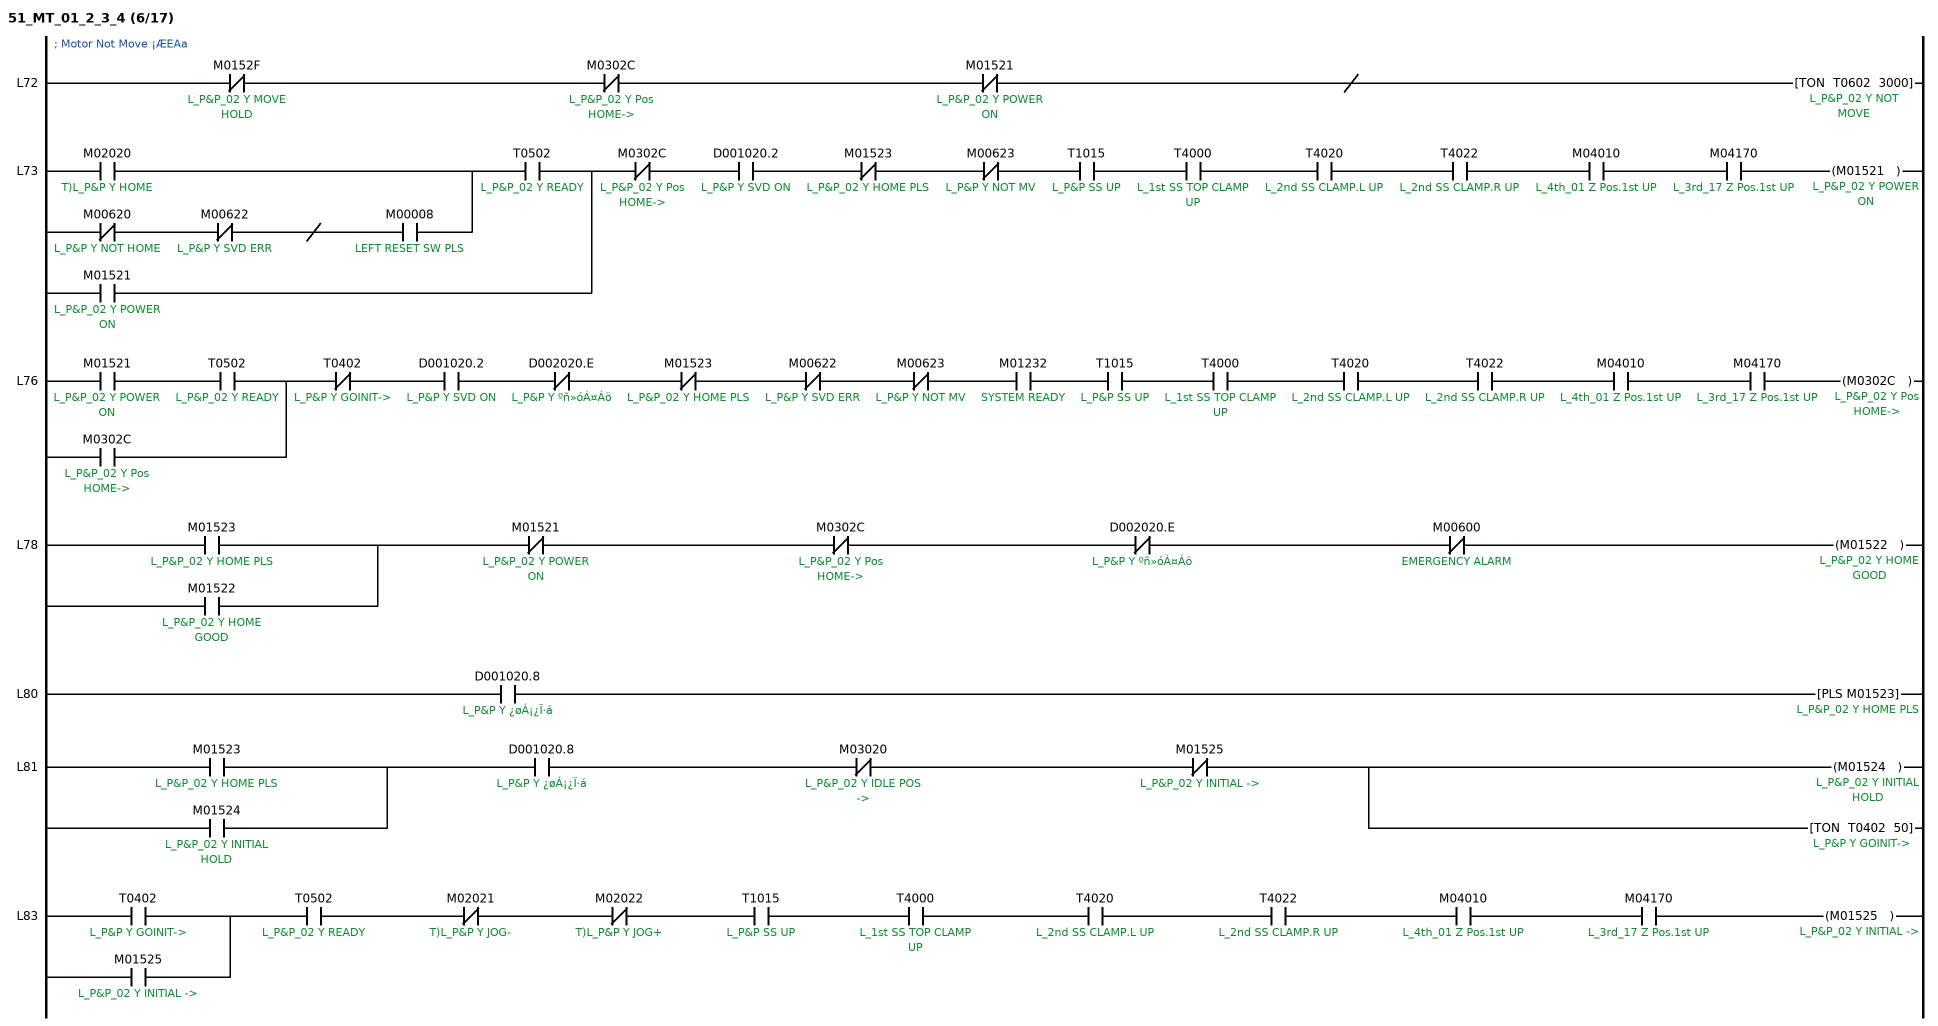
[picture p264: 51_MT_01_2_3_4 rungs L72-L83]
; L72
LOAD NOT  M0152F	// L_P&P_02 Y MOVE HOLD
AND NOT   M0302C	// L_P&P_02 Y Pos HOME->
AND NOT   M01521	// L_P&P_02 Y POWER ON
NOT
TON       T0602 3000	// L_P&P_02 Y NOT MOVE
// output comment: Motor Not Move ¡ÆEAa
; L73
LOAD      M02020	// T)L_P&P Y HOME
LOAD NOT  M00620	// L_P&P Y NOT HOME
AND NOT   M00622	// L_P&P Y SVD ERR
NOT
AND       M00008	// LEFT RESET SW PLS
OR LOAD
AND       T0502	// L_P&P_02 Y READY
OR        M01521	// L_P&P_02 Y POWER ON
AND NOT   M0302C	// L_P&P_02 Y Pos HOME->
AND       D001020.2	// L_P&P Y SVD ON
AND NOT   M01523	// L_P&P_02 Y HOME PLS
AND NOT   M00623	// L_P&P Y NOT MV
AND       T1015	// L_P&P SS UP
AND       T4000	// L_1st SS TOP CLAMP    UP
AND       T4020	// L_2nd SS CLAMP.L UP
AND       T4022	// L_2nd SS CLAMP.R UP
AND       M04010	// L_4th_01 Z Pos.1st UP
AND       M04170	// L_3rd_17 Z Pos.1st UP
OUT       M01521	// L_P&P_02 Y POWER ON
; L76
LOAD      M01521	// L_P&P_02 Y POWER ON
AND       T0502	// L_P&P_02 Y READY
OR        M0302C	// L_P&P_02 Y Pos HOME->
AND NOT   T0402	// L_P&P Y GOINIT->
AND       D001020.2	// L_P&P Y SVD ON
AND NOT   D002020.E	// L_P&P Y ºñ»óÁ¤Áö
AND NOT   M01523	// L_P&P_02 Y HOME PLS
AND NOT   M00622	// L_P&P Y SVD ERR
AND NOT   M00623	// L_P&P Y NOT MV
AND       M01232	// SYSTEM READY
AND       T1015	// L_P&P SS UP
AND       T4000	// L_1st SS TOP CLAMP    UP
AND       T4020	// L_2nd SS CLAMP.L UP
AND       T4022	// L_2nd SS CLAMP.R UP
AND       M04010	// L_4th_01 Z Pos.1st UP
AND       M04170	// L_3rd_17 Z Pos.1st UP
OUT       M0302C	// L_P&P_02 Y Pos HOME->
; L78
LOAD      M01523	// L_P&P_02 Y HOME PLS
OR        M01522	// L_P&P_02 Y HOME GOOD
AND NOT   M01521	// L_P&P_02 Y POWER ON
AND NOT   M0302C	// L_P&P_02 Y Pos HOME->
AND NOT   D002020.E	// L_P&P Y ºñ»óÁ¤Áö
AND NOT   M00600	// EMERGENCY ALARM
OUT       M01522	// L_P&P_02 Y HOME GOOD
; L80
LOAD      D001020.8	// L_P&P Y ¿øÁ¡¿Ï·á
OUTP      M01523	// L_P&P_02 Y HOME PLS
; L81
LOAD      M01523	// L_P&P_02 Y HOME PLS
OR        M01524	// L_P&P_02 Y INITIAL HOLD
AND       D001020.8	// L_P&P Y ¿øÁ¡¿Ï·á
AND NOT   M03020	// L_P&P_02 Y IDLE POS ->
AND NOT   M01525	// L_P&P_02 Y INITIAL ->
OUT       M01524	// L_P&P_02 Y INITIAL HOLD
TON       T0402 50	// L_P&P Y GOINIT->
; L83
LOAD      T0402	// L_P&P Y GOINIT->
OR        M01525	// L_P&P_02 Y INITIAL ->
AND       T0502	// L_P&P_02 Y READY
AND NOT   M02021	// T)L_P&P Y JOG-
AND NOT   M02022	// T)L_P&P Y JOG+
AND       T1015	// L_P&P SS UP
AND       T4000	// L_1st SS TOP CLAMP    UP
AND       T4020	// L_2nd SS CLAMP.L UP
AND       T4022	// L_2nd SS CLAMP.R UP
AND       M04010	// L_4th_01 Z Pos.1st UP
AND       M04170	// L_3rd_17 Z Pos.1st UP
OUT       M01525	// L_P&P_02 Y INITIAL ->

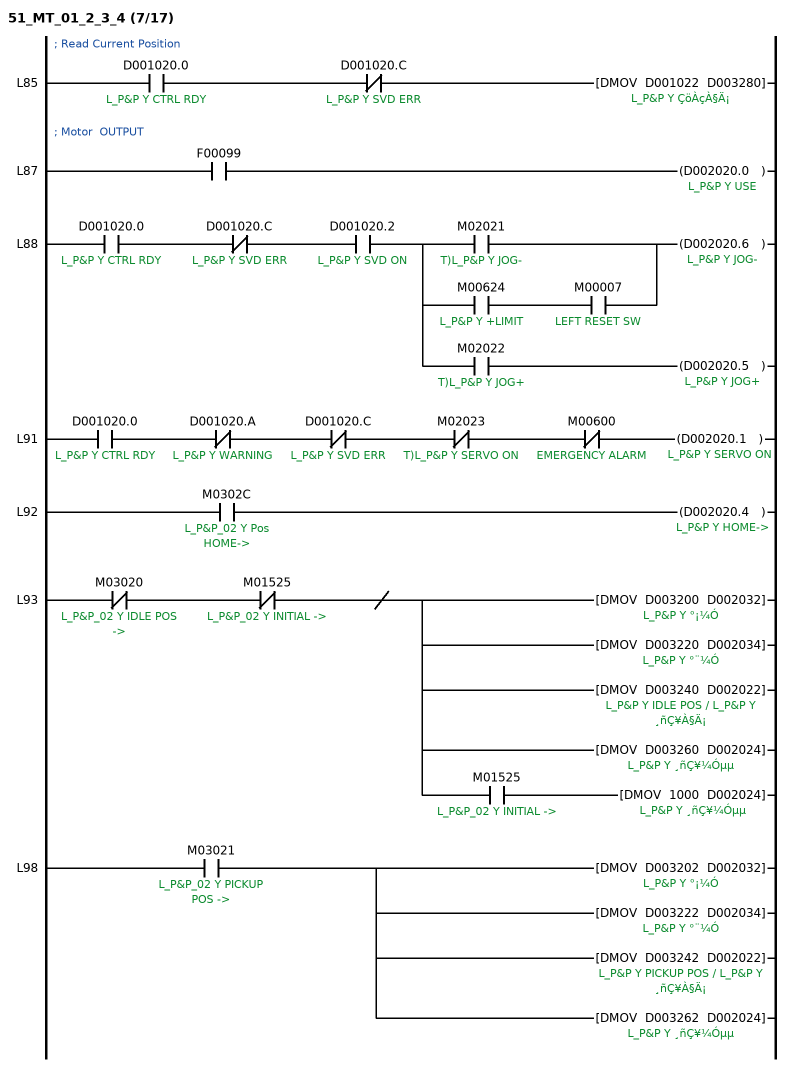
; L85
LOAD      D001020.0	// L_P&P Y CTRL RDY
AND NOT   D001020.C	// L_P&P Y SVD ERR
DMOV      D001022 D003280	// L_P&P Y ÇöÀçÀ§Ä¡
// output comment: Read Current Position
//  Motor  OUTPUT
; L87
LOAD      F00099
OUT       D002020.0	// L_P&P Y USE
; L88
LOAD      D001020.0	// L_P&P Y CTRL RDY
AND NOT   D001020.C	// L_P&P Y SVD ERR
AND       D001020.2	// L_P&P Y SVD ON
MPUSH
LOAD      M02021	// T)L_P&P Y JOG-
LOAD      M00624	// L_P&P Y +LIMIT
AND       M00007	// LEFT RESET SW
OR LOAD
AND LOAD
OUT       D002020.6	// L_P&P Y JOG-
MPOP
AND       M02022	// T)L_P&P Y JOG+
OUT       D002020.5	// L_P&P Y JOG+
; L91
LOAD      D001020.0	// L_P&P Y CTRL RDY
AND NOT   D001020.A	// L_P&P Y WARNING
AND NOT   D001020.C	// L_P&P Y SVD ERR
AND NOT   M02023	// T)L_P&P Y SERVO ON
AND NOT   M00600	// EMERGENCY ALARM
OUT       D002020.1	// L_P&P Y SERVO ON
; L92
LOAD      M0302C	// L_P&P_02 Y Pos HOME->
OUT       D002020.4	// L_P&P Y HOME->
; L93
LOAD NOT  M03020	// L_P&P_02 Y IDLE POS ->
AND NOT   M01525	// L_P&P_02 Y INITIAL ->
NOT
DMOV      D003200 D002032	// L_P&P Y °¡¼Ó
DMOV      D003220 D002034	// L_P&P Y °¨¼Ó
DMOV      D003240 D002022	// L_P&P Y IDLE POS / L_P&P Y ¸ñÇ¥À§Ä¡
DMOV      D003260 D002024	// L_P&P Y ¸ñÇ¥¼Óµµ
AND       M01525	// L_P&P_02 Y INITIAL ->
DMOV      1000 D002024	// L_P&P Y ¸ñÇ¥¼Óµµ
; L98
LOAD      M03021	// L_P&P_02 Y PICKUP POS ->
DMOV      D003202 D002032	// L_P&P Y °¡¼Ó
DMOV      D003222 D002034	// L_P&P Y °¨¼Ó
DMOV      D003242 D002022	// L_P&P Y PICKUP POS / L_P&P Y ¸ñÇ¥À§Ä¡
DMOV      D003262 D002024	// L_P&P Y ¸ñÇ¥¼Óµµ

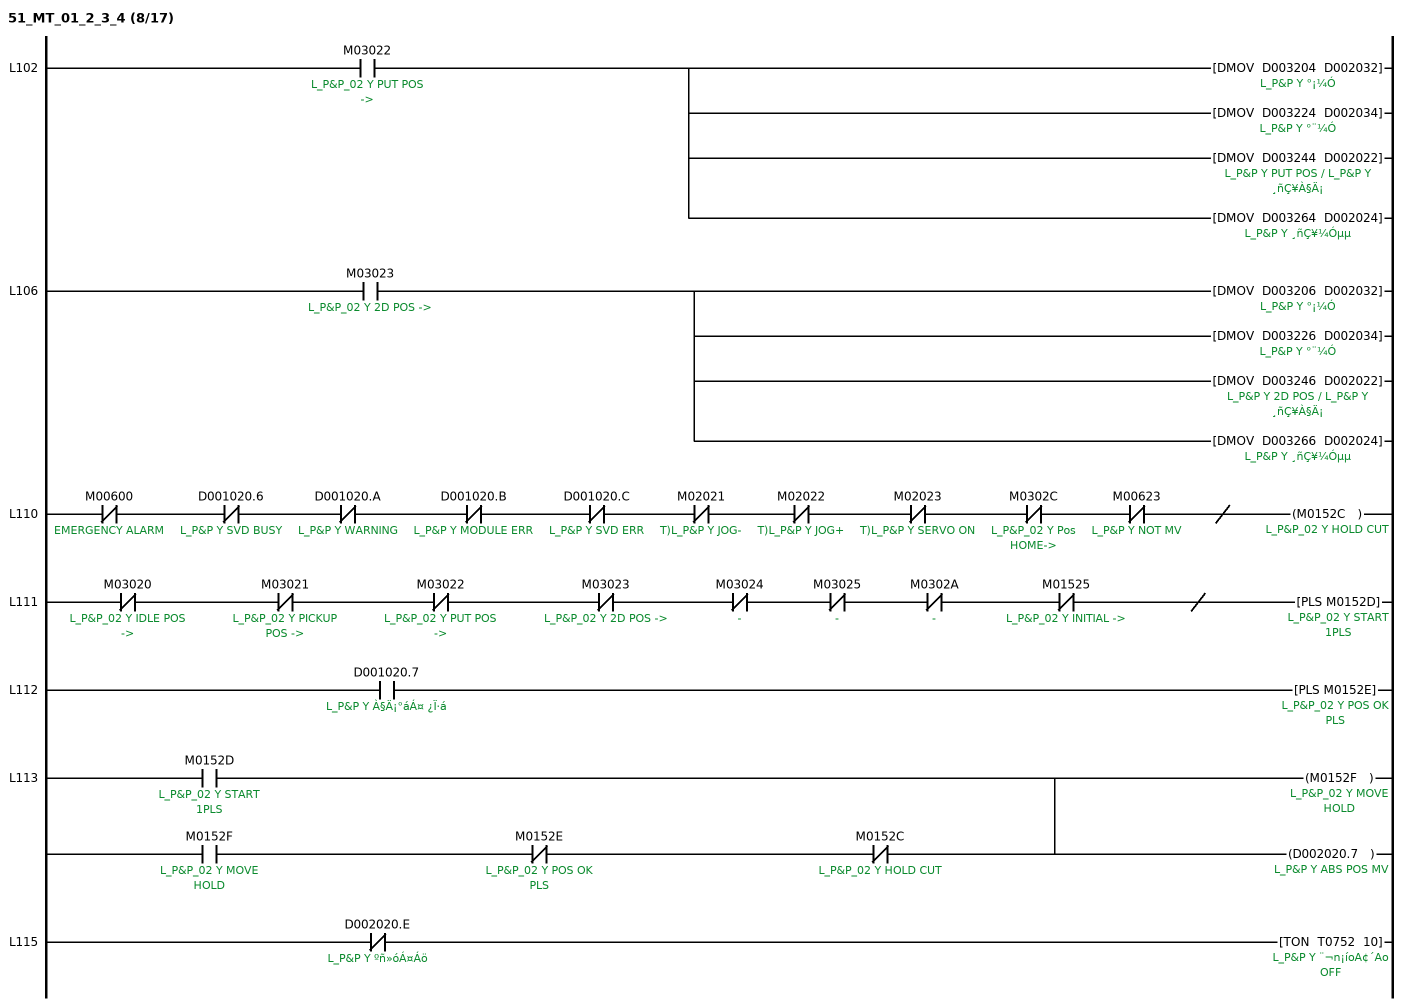
; L102
LOAD      M03022	// L_P&P_02 Y PUT POS ->
DMOV      D003204 D002032	// L_P&P Y °¡¼Ó
DMOV      D003224 D002034	// L_P&P Y °¨¼Ó
DMOV      D003244 D002022	// L_P&P Y PUT POS / L_P&P Y ¸ñÇ¥À§Ä¡
DMOV      D003264 D002024	// L_P&P Y ¸ñÇ¥¼Óµµ
; L106
LOAD      M03023	// L_P&P_02 Y 2D POS ->
DMOV      D003206 D002032	// L_P&P Y °¡¼Ó
DMOV      D003226 D002034	// L_P&P Y °¨¼Ó
DMOV      D003246 D002022	// L_P&P Y 2D POS / L_P&P Y ¸ñÇ¥À§Ä¡
DMOV      D003266 D002024	// L_P&P Y ¸ñÇ¥¼Óµµ
; L110
LOAD NOT  M00600	// EMERGENCY ALARM
AND NOT   D001020.6	// L_P&P Y SVD BUSY
AND NOT   D001020.A	// L_P&P Y WARNING
AND NOT   D001020.B	// L_P&P Y MODULE ERR
AND NOT   D001020.C	// L_P&P Y SVD ERR
AND NOT   M02021	// T)L_P&P Y JOG-
AND NOT   M02022	// T)L_P&P Y JOG+
AND NOT   M02023	// T)L_P&P Y SERVO ON
AND NOT   M0302C	// L_P&P_02 Y Pos HOME->
AND NOT   M00623	// L_P&P Y NOT MV
NOT
OUT       M0152C	// L_P&P_02 Y HOLD CUT
; L111
LOAD NOT  M03020	// L_P&P_02 Y IDLE POS ->
AND NOT   M03021	// L_P&P_02 Y PICKUP POS ->
AND NOT   M03022	// L_P&P_02 Y PUT POS ->
AND NOT   M03023	// L_P&P_02 Y 2D POS ->
AND NOT   M03024	// -
AND NOT   M03025	// -
AND NOT   M0302A	// -
AND NOT   M01525	// L_P&P_02 Y INITIAL ->
NOT
OUTP      M0152D	// L_P&P_02 Y START 1PLS
; L112
LOAD      D001020.7	// L_P&P Y À§Ä¡°áÁ¤ ¿Ï·á
OUTP      M0152E	// L_P&P_02 Y POS OK PLS
; L113
LOAD      M0152D	// L_P&P_02 Y START 1PLS
LOAD      M0152F	// L_P&P_02 Y MOVE HOLD
AND NOT   M0152E	// L_P&P_02 Y POS OK PLS
AND NOT   M0152C	// L_P&P_02 Y HOLD CUT
OR LOAD
OUT       M0152F	// L_P&P_02 Y MOVE HOLD
OUT       D002020.7	// L_P&P Y ABS POS MV
; L115
LOAD NOT  D002020.E	// L_P&P Y ºñ»óÁ¤Áö
TON       T0752 10	// L_P&P Y ¨¬n¡íoA¢´AoOFF

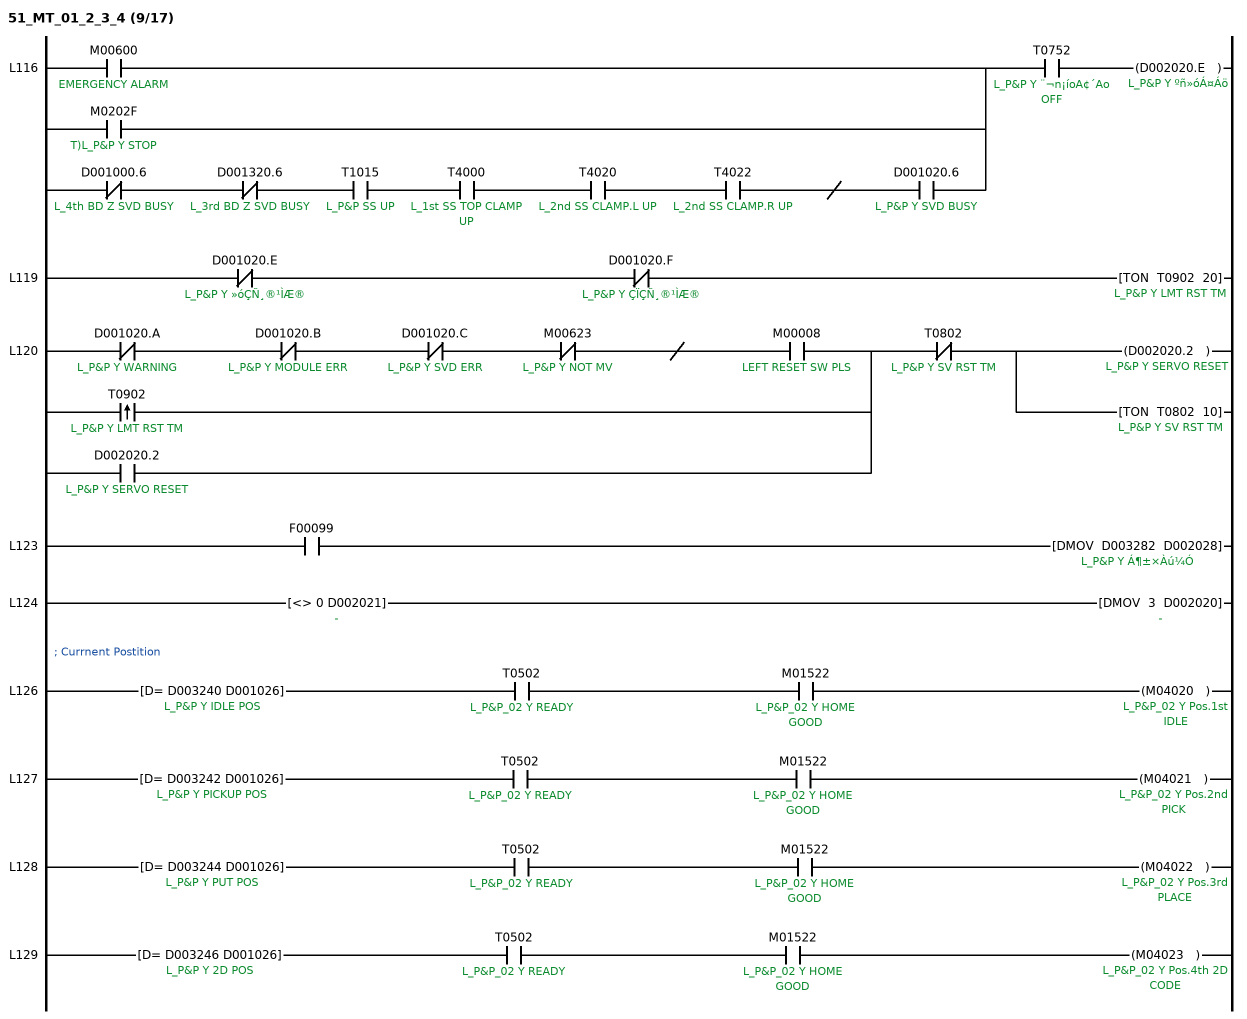
; L116
LOAD      M00600	// EMERGENCY ALARM
OR        M0202F	// T)L_P&P Y STOP
LOAD NOT  D001000.6	// L_4th BD Z SVD BUSY
AND NOT   D001320.6	// L_3rd BD Z SVD BUSY
AND       T1015	// L_P&P SS UP
AND       T4000	// L_1st SS TOP CLAMP    UP
AND       T4020	// L_2nd SS CLAMP.L UP
AND       T4022	// L_2nd SS CLAMP.R UP
NOT
AND       D001020.6	// L_P&P Y SVD BUSY
OR LOAD
AND       T0752	// L_P&P Y ¨¬n¡íoA¢´AoOFF
OUT       D002020.E	// L_P&P Y ºñ»óÁ¤Áö
; L119
LOAD NOT  D001020.E	// L_P&P Y »óÇÑ¸®¹ÌÆ®
AND NOT   D001020.F	// L_P&P Y ÇÏÇÑ¸®¹ÌÆ®
TON       T0902 20	// L_P&P Y LMT RST TM
; L120
LOAD NOT  D001020.A	// L_P&P Y WARNING
AND NOT   D001020.B	// L_P&P Y MODULE ERR
AND NOT   D001020.C	// L_P&P Y SVD ERR
AND NOT   M00623	// L_P&P Y NOT MV
NOT
AND       M00008	// LEFT RESET SW PLS
ORP       T0902	// L_P&P Y LMT RST TM
OR        D002020.2	// L_P&P Y SERVO RESET
AND NOT   T0802	// L_P&P Y SV RST TM
OUT       D002020.2	// L_P&P Y SERVO RESET
TON       T0802 10	// L_P&P Y SV RST TM
; L123
LOAD      F00099
DMOV      D003282 D002028	// L_P&P Y Á¶±×Àú¼Ó
; L124
LOAD<>    0 D002021	// -
DMOV      3 D002020	// -
// Currnent Postition
; L126
LOADD=    D003240 D001026	// L_P&P Y IDLE POS
AND       T0502	// L_P&P_02 Y READY
AND       M01522	// L_P&P_02 Y HOME GOOD
OUT       M04020	// L_P&P_02 Y Pos.1st IDLE
; L127
LOADD=    D003242 D001026	// L_P&P Y PICKUP POS
AND       T0502	// L_P&P_02 Y READY
AND       M01522	// L_P&P_02 Y HOME GOOD
OUT       M04021	// L_P&P_02 Y Pos.2nd PICK
; L128
LOADD=    D003244 D001026	// L_P&P Y PUT POS
AND       T0502	// L_P&P_02 Y READY
AND       M01522	// L_P&P_02 Y HOME GOOD
OUT       M04022	// L_P&P_02 Y Pos.3rd PLACE
; L129
LOADD=    D003246 D001026	// L_P&P Y 2D POS
AND       T0502	// L_P&P_02 Y READY
AND       M01522	// L_P&P_02 Y HOME GOOD
OUT       M04023	// L_P&P_02 Y Pos.4th 2D CODE

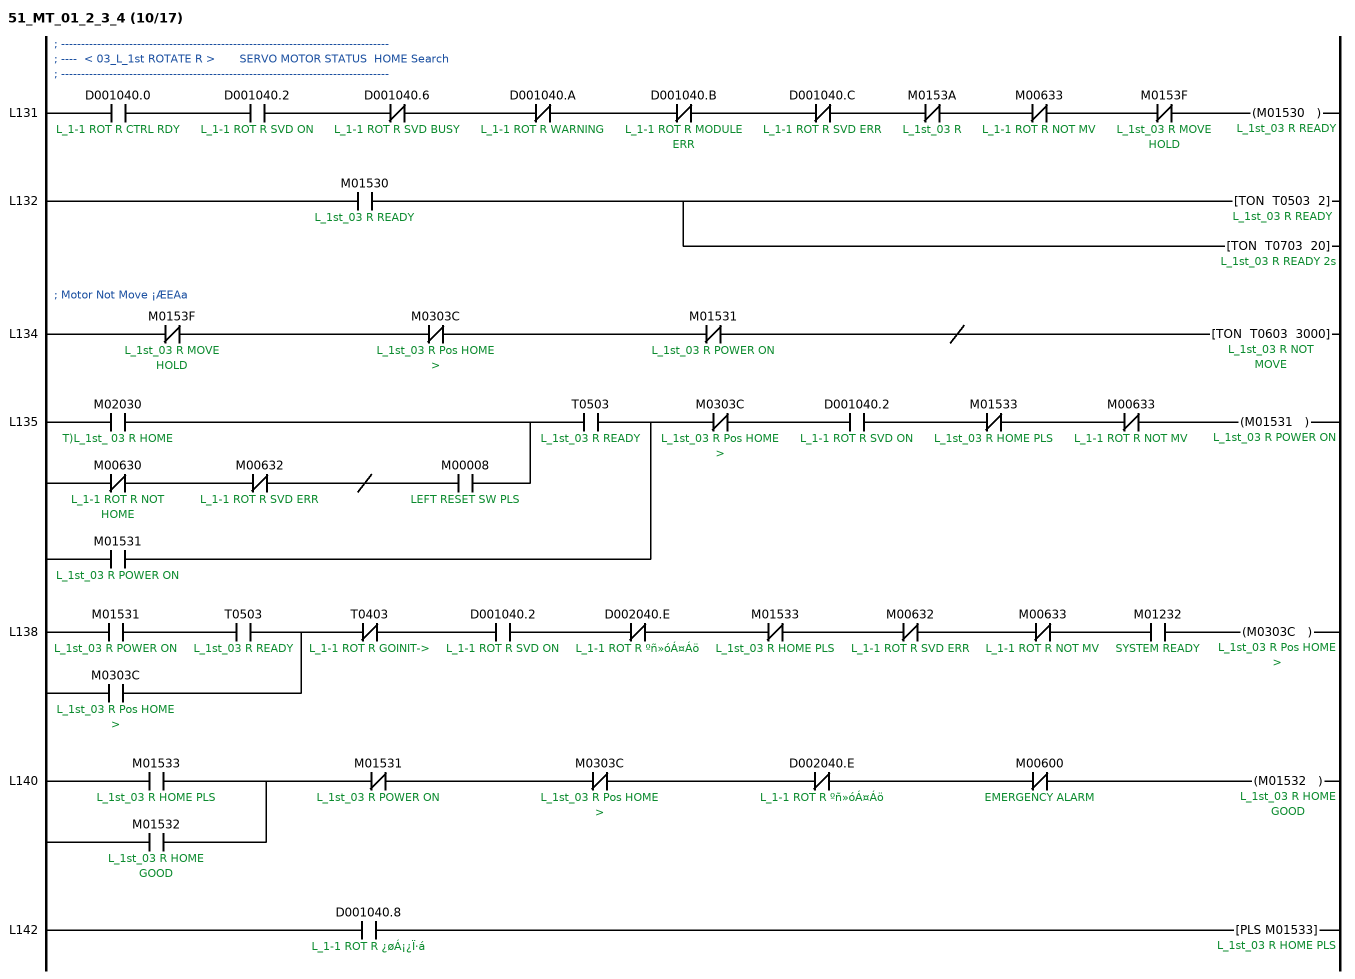
// ----------------------------------------------------------------------------------
// 
// ----  < 03_L_1st ROTATE R >       SERVO MOTOR STATUS  HOME Search
// 
// ----------------------------------------------------------------------------------
; L131
LOAD      D001040.0	// L_1-1 ROT R CTRL RDY
AND       D001040.2	// L_1-1 ROT R SVD ON
AND NOT   D001040.6	// L_1-1 ROT R SVD BUSY
AND NOT   D001040.A	// L_1-1 ROT R WARNING
AND NOT   D001040.B	// L_1-1 ROT R MODULE ERR
AND NOT   D001040.C	// L_1-1 ROT R SVD ERR
AND NOT   M0153A	// L_1st_03 R
AND NOT   M00633	// L_1-1 ROT R NOT MV
AND NOT   M0153F	// L_1st_03 R MOVE HOLD
OUT       M01530	// L_1st_03 R READY
; L132
LOAD      M01530	// L_1st_03 R READY
TON       T0503 2	// L_1st_03 R READY
TON       T0703 20	// L_1st_03 R READY 2s
; L134
LOAD NOT  M0153F	// L_1st_03 R MOVE HOLD
AND NOT   M0303C	// L_1st_03 R Pos HOME >
AND NOT   M01531	// L_1st_03 R POWER ON
NOT
TON       T0603 3000	// L_1st_03 R NOT MOVE
// output comment: Motor Not Move ¡ÆEAa
; L135
LOAD      M02030	// T)L_1st_ 03 R HOME
LOAD NOT  M00630	// L_1-1 ROT R NOT HOME
AND NOT   M00632	// L_1-1 ROT R SVD ERR
NOT
AND       M00008	// LEFT RESET SW PLS
OR LOAD
AND       T0503	// L_1st_03 R READY
OR        M01531	// L_1st_03 R POWER ON
AND NOT   M0303C	// L_1st_03 R Pos HOME >
AND       D001040.2	// L_1-1 ROT R SVD ON
AND NOT   M01533	// L_1st_03 R HOME PLS
AND NOT   M00633	// L_1-1 ROT R NOT MV
OUT       M01531	// L_1st_03 R POWER ON
; L138
LOAD      M01531	// L_1st_03 R POWER ON
AND       T0503	// L_1st_03 R READY
OR        M0303C	// L_1st_03 R Pos HOME >
AND NOT   T0403	// L_1-1 ROT R GOINIT->
AND       D001040.2	// L_1-1 ROT R SVD ON
AND NOT   D002040.E	// L_1-1 ROT R ºñ»óÁ¤Áö
AND NOT   M01533	// L_1st_03 R HOME PLS
AND NOT   M00632	// L_1-1 ROT R SVD ERR
AND NOT   M00633	// L_1-1 ROT R NOT MV
AND       M01232	// SYSTEM READY
OUT       M0303C	// L_1st_03 R Pos HOME >
; L140
LOAD      M01533	// L_1st_03 R HOME PLS
OR        M01532	// L_1st_03 R HOME GOOD
AND NOT   M01531	// L_1st_03 R POWER ON
AND NOT   M0303C	// L_1st_03 R Pos HOME >
AND NOT   D002040.E	// L_1-1 ROT R ºñ»óÁ¤Áö
AND NOT   M00600	// EMERGENCY ALARM
OUT       M01532	// L_1st_03 R HOME GOOD
; L142
LOAD      D001040.8	// L_1-1 ROT R ¿øÁ¡¿Ï·á
OUTP      M01533	// L_1st_03 R HOME PLS

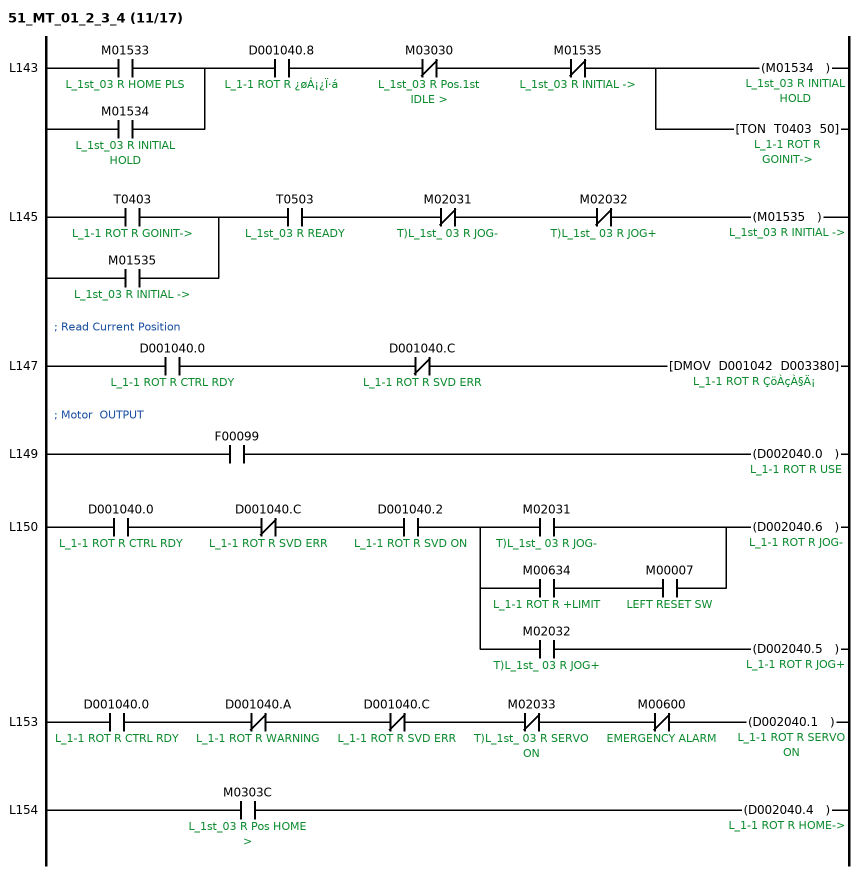
; L143
LOAD      M01533	// L_1st_03 R HOME PLS
OR        M01534	// L_1st_03 R INITIAL HOLD
AND       D001040.8	// L_1-1 ROT R ¿øÁ¡¿Ï·á
AND NOT   M03030	// L_1st_03 R Pos.1st IDLE >
AND NOT   M01535	// L_1st_03 R INITIAL ->
OUT       M01534	// L_1st_03 R INITIAL HOLD
TON       T0403 50	// L_1-1 ROT R GOINIT->
; L145
LOAD      T0403	// L_1-1 ROT R GOINIT->
OR        M01535	// L_1st_03 R INITIAL ->
AND       T0503	// L_1st_03 R READY
AND NOT   M02031	// T)L_1st_ 03 R JOG-
AND NOT   M02032	// T)L_1st_ 03 R JOG+
OUT       M01535	// L_1st_03 R INITIAL ->
; L147
LOAD      D001040.0	// L_1-1 ROT R CTRL RDY
AND NOT   D001040.C	// L_1-1 ROT R SVD ERR
DMOV      D001042 D003380	// L_1-1 ROT R ÇöÀçÀ§Ä¡
// output comment: Read Current Position
//  Motor  OUTPUT
; L149
LOAD      F00099
OUT       D002040.0	// L_1-1 ROT R USE
; L150
LOAD      D001040.0	// L_1-1 ROT R CTRL RDY
AND NOT   D001040.C	// L_1-1 ROT R SVD ERR
AND       D001040.2	// L_1-1 ROT R SVD ON
MPUSH
LOAD      M02031	// T)L_1st_ 03 R JOG-
LOAD      M00634	// L_1-1 ROT R +LIMIT
AND       M00007	// LEFT RESET SW
OR LOAD
AND LOAD
OUT       D002040.6	// L_1-1 ROT R JOG-
MPOP
AND       M02032	// T)L_1st_ 03 R JOG+
OUT       D002040.5	// L_1-1 ROT R JOG+
; L153
LOAD      D001040.0	// L_1-1 ROT R CTRL RDY
AND NOT   D001040.A	// L_1-1 ROT R WARNING
AND NOT   D001040.C	// L_1-1 ROT R SVD ERR
AND NOT   M02033	// T)L_1st_ 03 R SERVO ON
AND NOT   M00600	// EMERGENCY ALARM
OUT       D002040.1	// L_1-1 ROT R SERVO ON
; L154
LOAD      M0303C	// L_1st_03 R Pos HOME >
OUT       D002040.4	// L_1-1 ROT R HOME->

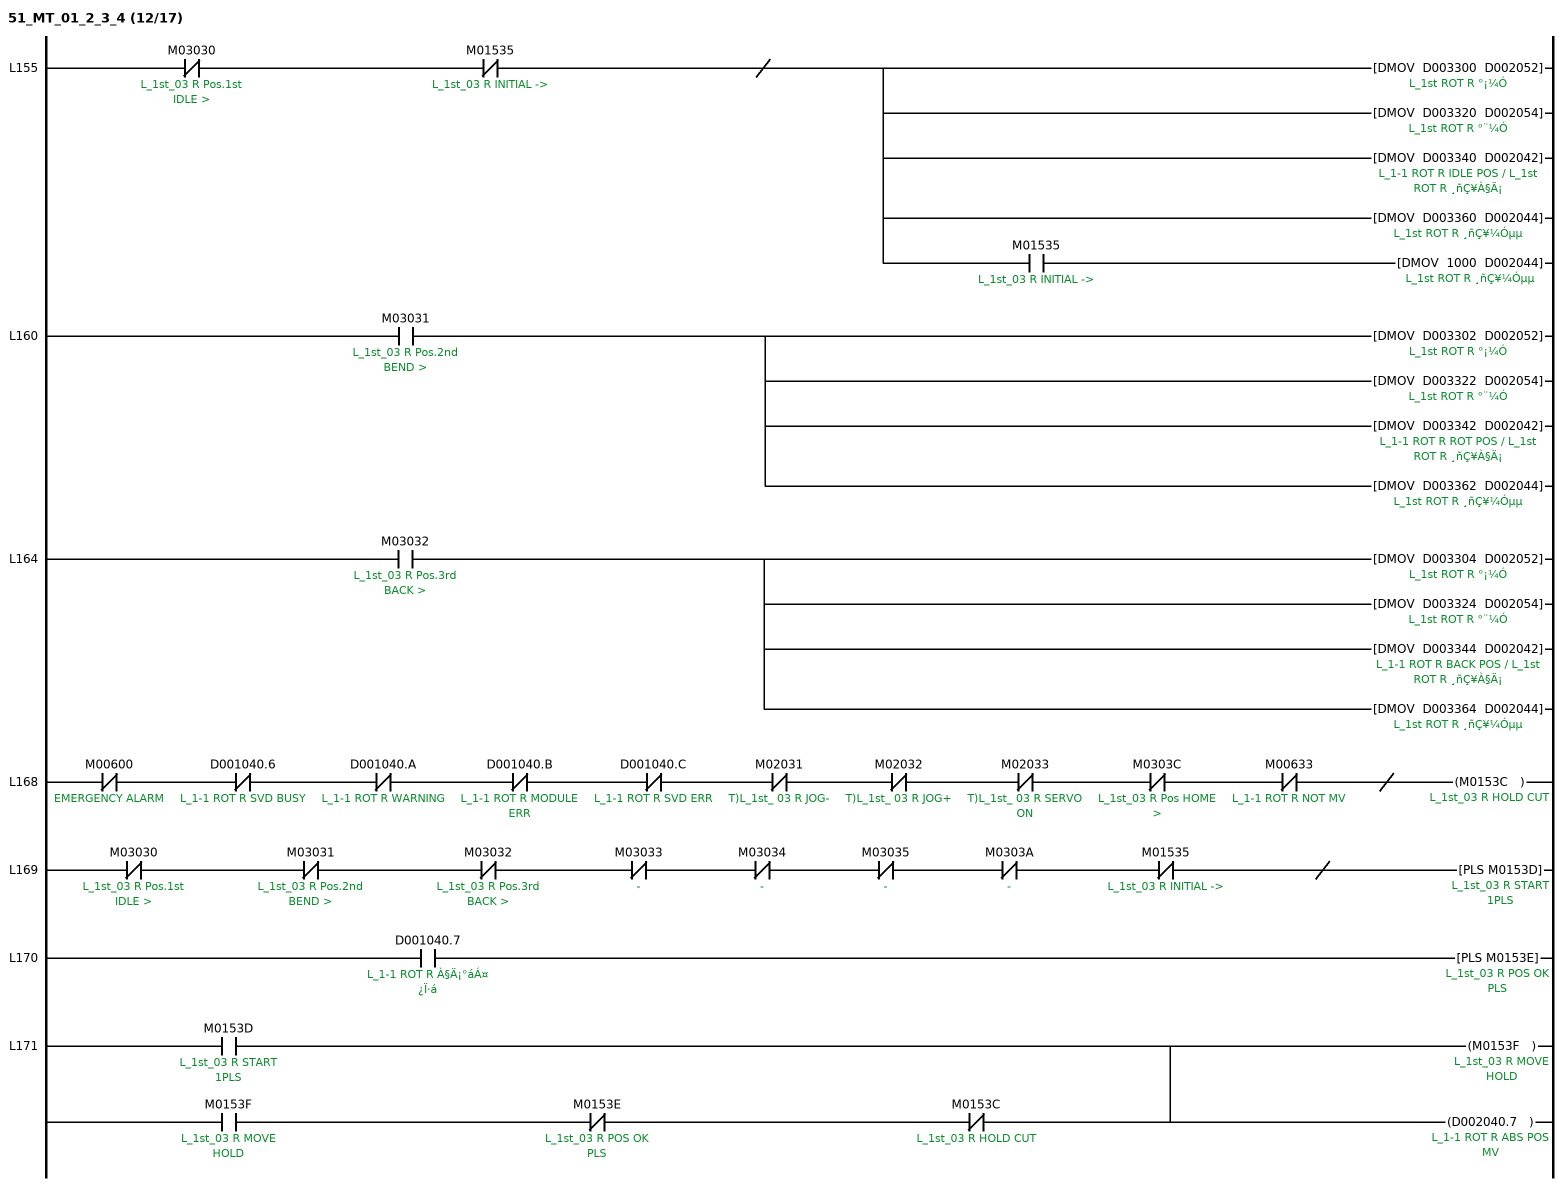
; L155
LOAD NOT  M03030	// L_1st_03 R Pos.1st IDLE >
AND NOT   M01535	// L_1st_03 R INITIAL ->
NOT
DMOV      D003300 D002052	// L_1st ROT R °¡¼Ó
DMOV      D003320 D002054	// L_1st ROT R °¨¼Ó
DMOV      D003340 D002042	// L_1-1 ROT R IDLE POS / L_1st ROT R ¸ñÇ¥À§Ä¡
DMOV      D003360 D002044	// L_1st ROT R ¸ñÇ¥¼Óµµ
AND       M01535	// L_1st_03 R INITIAL ->
DMOV      1000 D002044	// L_1st ROT R ¸ñÇ¥¼Óµµ
; L160
LOAD      M03031	// L_1st_03 R Pos.2nd BEND >
DMOV      D003302 D002052	// L_1st ROT R °¡¼Ó
DMOV      D003322 D002054	// L_1st ROT R °¨¼Ó
DMOV      D003342 D002042	// L_1-1 ROT R ROT POS / L_1st ROT R ¸ñÇ¥À§Ä¡
DMOV      D003362 D002044	// L_1st ROT R ¸ñÇ¥¼Óµµ
; L164
LOAD      M03032	// L_1st_03 R Pos.3rd BACK >
DMOV      D003304 D002052	// L_1st ROT R °¡¼Ó
DMOV      D003324 D002054	// L_1st ROT R °¨¼Ó
DMOV      D003344 D002042	// L_1-1 ROT R BACK POS / L_1st ROT R ¸ñÇ¥À§Ä¡
DMOV      D003364 D002044	// L_1st ROT R ¸ñÇ¥¼Óµµ
; L168
LOAD NOT  M00600	// EMERGENCY ALARM
AND NOT   D001040.6	// L_1-1 ROT R SVD BUSY
AND NOT   D001040.A	// L_1-1 ROT R WARNING
AND NOT   D001040.B	// L_1-1 ROT R MODULE ERR
AND NOT   D001040.C	// L_1-1 ROT R SVD ERR
AND NOT   M02031	// T)L_1st_ 03 R JOG-
AND NOT   M02032	// T)L_1st_ 03 R JOG+
AND NOT   M02033	// T)L_1st_ 03 R SERVO ON
AND NOT   M0303C	// L_1st_03 R Pos HOME >
AND NOT   M00633	// L_1-1 ROT R NOT MV
NOT
OUT       M0153C	// L_1st_03 R HOLD CUT
; L169
LOAD NOT  M03030	// L_1st_03 R Pos.1st IDLE >
AND NOT   M03031	// L_1st_03 R Pos.2nd BEND >
AND NOT   M03032	// L_1st_03 R Pos.3rd BACK >
AND NOT   M03033	// -
AND NOT   M03034	// -
AND NOT   M03035	// -
AND NOT   M0303A	// -
AND NOT   M01535	// L_1st_03 R INITIAL ->
NOT
OUTP      M0153D	// L_1st_03 R START 1PLS
; L170
LOAD      D001040.7	// L_1-1 ROT R À§Ä¡°áÁ¤ ¿Ï·á
OUTP      M0153E	// L_1st_03 R POS OK PLS
; L171
LOAD      M0153D	// L_1st_03 R START 1PLS
LOAD      M0153F	// L_1st_03 R MOVE HOLD
AND NOT   M0153E	// L_1st_03 R POS OK PLS
AND NOT   M0153C	// L_1st_03 R HOLD CUT
OR LOAD
OUT       M0153F	// L_1st_03 R MOVE HOLD
OUT       D002040.7	// L_1-1 ROT R ABS POS MV

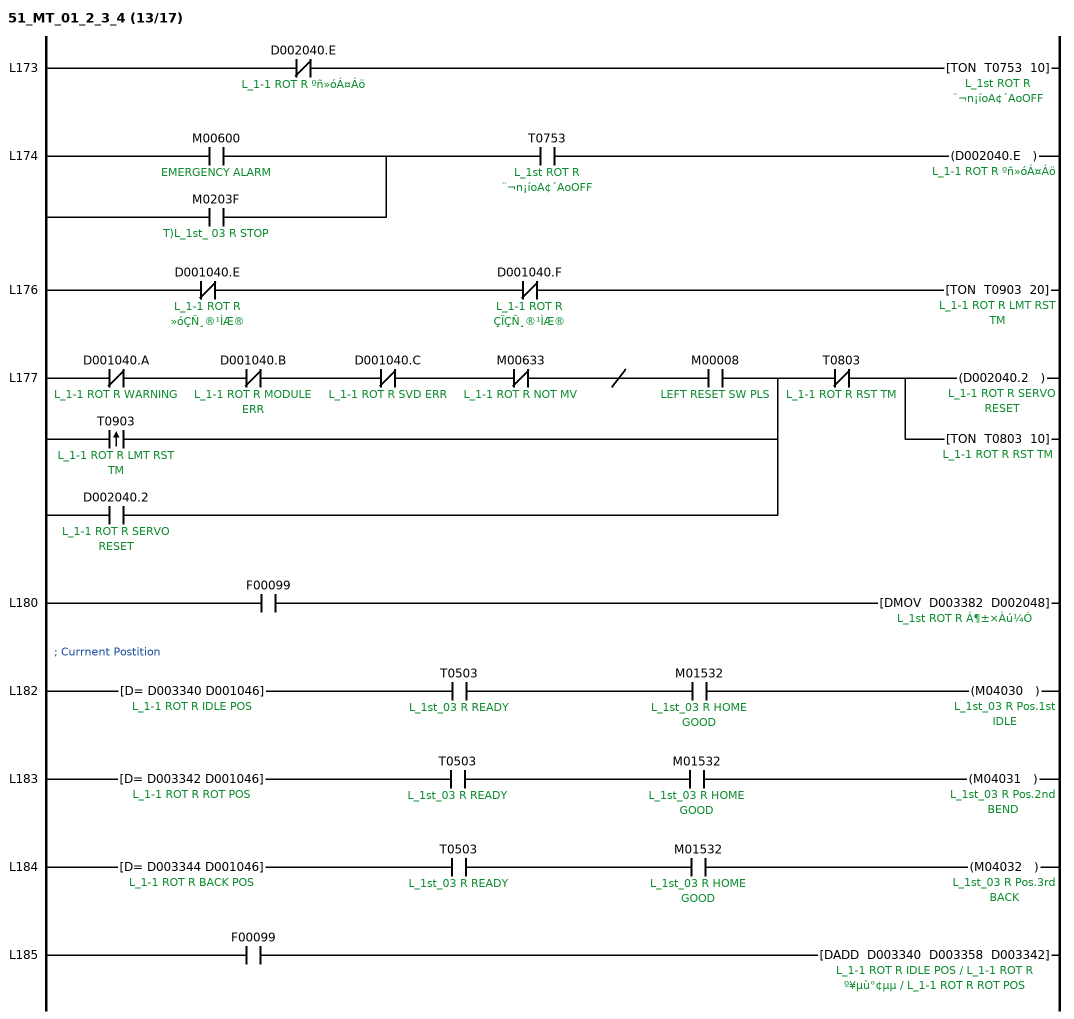
; L173
LOAD NOT  D002040.E	// L_1-1 ROT R ºñ»óÁ¤Áö
TON       T0753 10	// L_1st ROT R ¨¬n¡íoA¢´AoOFF
; L174
LOAD      M00600	// EMERGENCY ALARM
OR        M0203F	// T)L_1st_ 03 R STOP
AND       T0753	// L_1st ROT R ¨¬n¡íoA¢´AoOFF
OUT       D002040.E	// L_1-1 ROT R ºñ»óÁ¤Áö
; L176
LOAD NOT  D001040.E	// L_1-1 ROT R »óÇÑ¸®¹ÌÆ®
AND NOT   D001040.F	// L_1-1 ROT R ÇÏÇÑ¸®¹ÌÆ®
TON       T0903 20	// L_1-1 ROT R LMT RST TM
; L177
LOAD NOT  D001040.A	// L_1-1 ROT R WARNING
AND NOT   D001040.B	// L_1-1 ROT R MODULE ERR
AND NOT   D001040.C	// L_1-1 ROT R SVD ERR
AND NOT   M00633	// L_1-1 ROT R NOT MV
NOT
AND       M00008	// LEFT RESET SW PLS
ORP       T0903	// L_1-1 ROT R LMT RST TM
OR        D002040.2	// L_1-1 ROT R SERVO RESET
AND NOT   T0803	// L_1-1 ROT R RST TM
OUT       D002040.2	// L_1-1 ROT R SERVO RESET
TON       T0803 10	// L_1-1 ROT R RST TM
; L180
LOAD      F00099
DMOV      D003382 D002048	// L_1st ROT R Á¶±×Àú¼Ó
// Currnent Postition
; L182
LOADD=    D003340 D001046	// L_1-1 ROT R IDLE POS
AND       T0503	// L_1st_03 R READY
AND       M01532	// L_1st_03 R HOME GOOD
OUT       M04030	// L_1st_03 R Pos.1st IDLE
; L183
LOADD=    D003342 D001046	// L_1-1 ROT R ROT POS
AND       T0503	// L_1st_03 R READY
AND       M01532	// L_1st_03 R HOME GOOD
OUT       M04031	// L_1st_03 R Pos.2nd BEND
; L184
LOADD=    D003344 D001046	// L_1-1 ROT R BACK POS
AND       T0503	// L_1st_03 R READY
AND       M01532	// L_1st_03 R HOME GOOD
OUT       M04032	// L_1st_03 R Pos.3rd BACK
; L185
LOAD      F00099
DADD      D003340 D003358 D003342	// L_1-1 ROT R IDLE POS / L_1-1 ROT R º¥µù°¢µµ / L_1-1 ROT R ROT POS

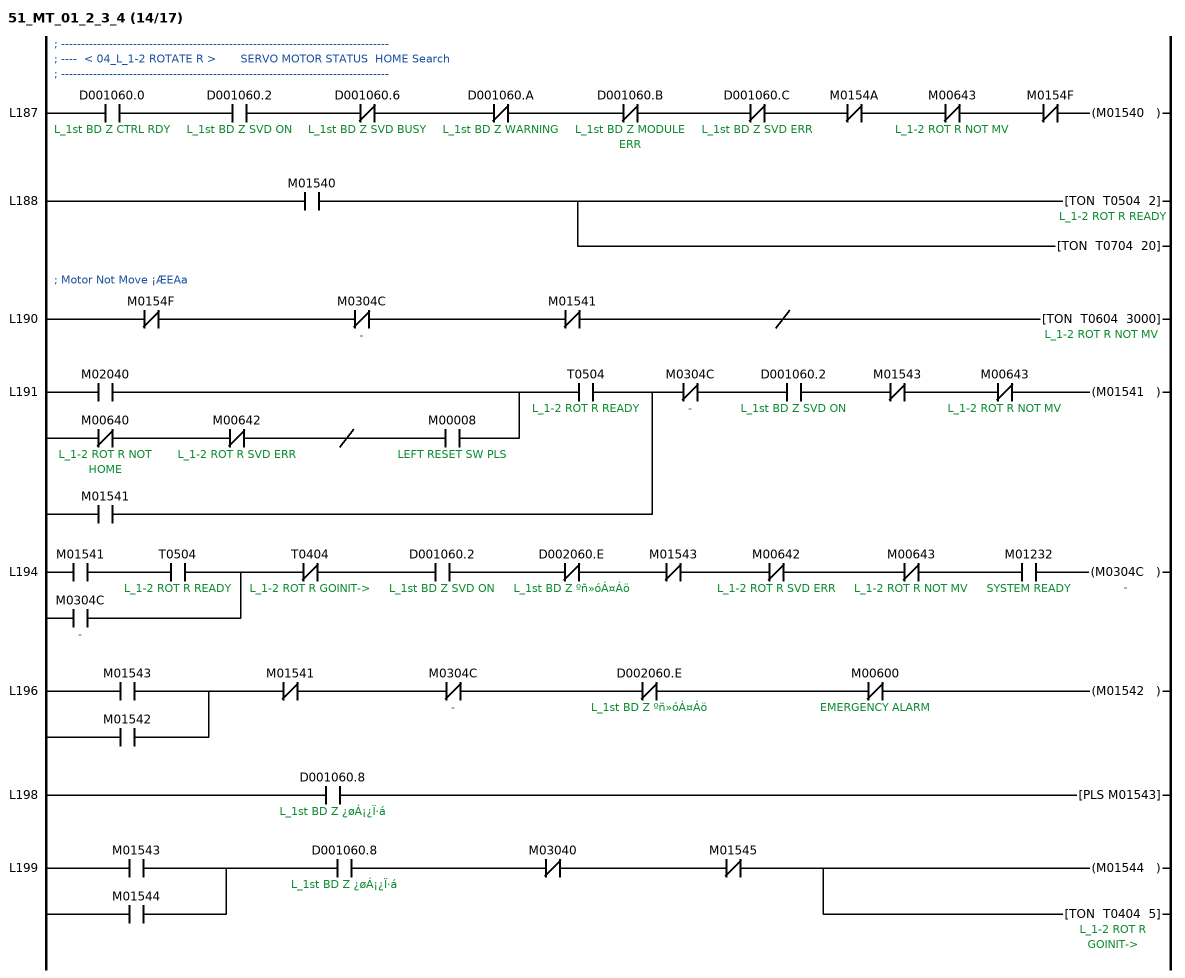
// ----------------------------------------------------------------------------------
// 
// ----  < 04_L_1-2 ROTATE R >       SERVO MOTOR STATUS  HOME Search
// 
// ----------------------------------------------------------------------------------
; L187
LOAD      D001060.0	// L_1st BD Z CTRL RDY
AND       D001060.2	// L_1st BD Z SVD ON
AND NOT   D001060.6	// L_1st BD Z SVD BUSY
AND NOT   D001060.A	// L_1st BD Z WARNING
AND NOT   D001060.B	// L_1st BD Z MODULE ERR
AND NOT   D001060.C	// L_1st BD Z SVD ERR
AND NOT   M0154A
AND NOT   M00643	// L_1-2 ROT R NOT MV
AND NOT   M0154F
OUT       M01540
; L188
LOAD      M01540
TON       T0504 2	// L_1-2 ROT R READY
TON       T0704 20
; L190
LOAD NOT  M0154F
AND NOT   M0304C	// -
AND NOT   M01541
NOT
TON       T0604 3000	// L_1-2 ROT R NOT MV
// output comment: Motor Not Move ¡ÆEAa
; L191
LOAD      M02040
LOAD NOT  M00640	// L_1-2 ROT R NOT HOME
AND NOT   M00642	// L_1-2 ROT R SVD ERR
NOT
AND       M00008	// LEFT RESET SW PLS
OR LOAD
AND       T0504	// L_1-2 ROT R READY
OR        M01541
AND NOT   M0304C	// -
AND       D001060.2	// L_1st BD Z SVD ON
AND NOT   M01543
AND NOT   M00643	// L_1-2 ROT R NOT MV
OUT       M01541
; L194
LOAD      M01541
AND       T0504	// L_1-2 ROT R READY
OR        M0304C	// -
AND NOT   T0404	// L_1-2 ROT R GOINIT->
AND       D001060.2	// L_1st BD Z SVD ON
AND NOT   D002060.E	// L_1st BD Z ºñ»óÁ¤Áö
AND NOT   M01543
AND NOT   M00642	// L_1-2 ROT R SVD ERR
AND NOT   M00643	// L_1-2 ROT R NOT MV
AND       M01232	// SYSTEM READY
OUT       M0304C	// -
; L196
LOAD      M01543
OR        M01542
AND NOT   M01541
AND NOT   M0304C	// -
AND NOT   D002060.E	// L_1st BD Z ºñ»óÁ¤Áö
AND NOT   M00600	// EMERGENCY ALARM
OUT       M01542
; L198
LOAD      D001060.8	// L_1st BD Z ¿øÁ¡¿Ï·á
OUTP      M01543
; L199
LOAD      M01543
OR        M01544
AND       D001060.8	// L_1st BD Z ¿øÁ¡¿Ï·á
AND NOT   M03040
AND NOT   M01545
OUT       M01544
TON       T0404 5	// L_1-2 ROT R GOINIT->

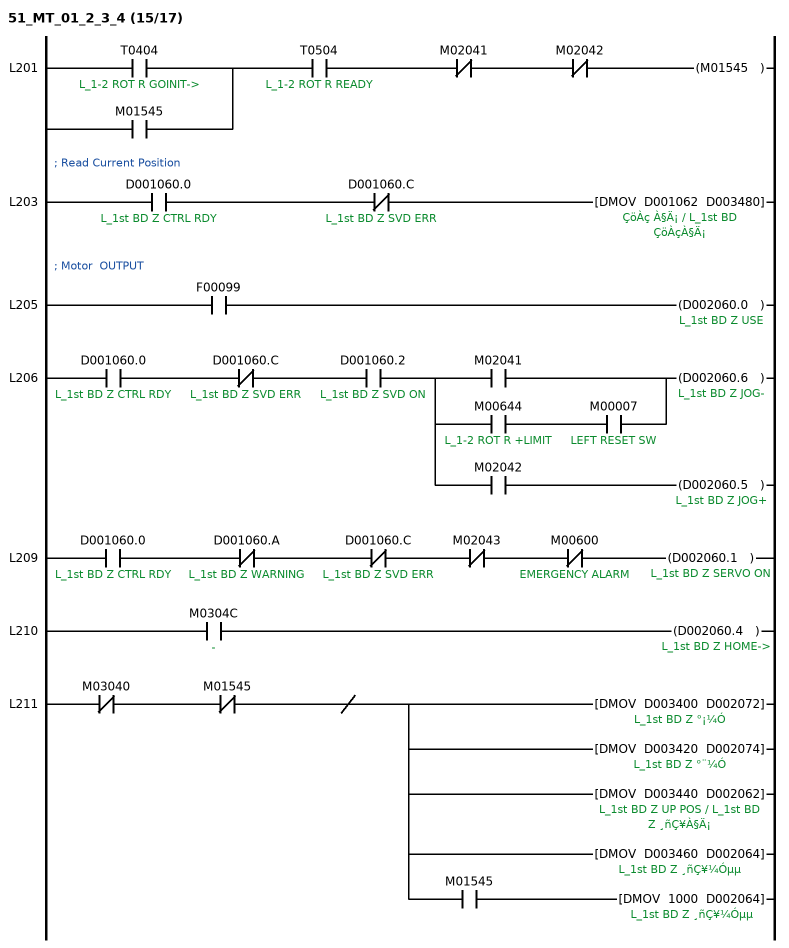
; L201
LOAD      T0404	// L_1-2 ROT R GOINIT->
OR        M01545
AND       T0504	// L_1-2 ROT R READY
AND NOT   M02041
AND NOT   M02042
OUT       M01545
; L203
LOAD      D001060.0	// L_1st BD Z CTRL RDY
AND NOT   D001060.C	// L_1st BD Z SVD ERR
DMOV      D001062 D003480	// ÇöÀç À§Ä¡ / L_1st BD ÇöÀçÀ§Ä¡
// output comment: Read Current Position
//  Motor  OUTPUT
; L205
LOAD      F00099
OUT       D002060.0	// L_1st BD Z USE
; L206
LOAD      D001060.0	// L_1st BD Z CTRL RDY
AND NOT   D001060.C	// L_1st BD Z SVD ERR
AND       D001060.2	// L_1st BD Z SVD ON
MPUSH
LOAD      M02041
LOAD      M00644	// L_1-2 ROT R +LIMIT
AND       M00007	// LEFT RESET SW
OR LOAD
AND LOAD
OUT       D002060.6	// L_1st BD Z JOG-
MPOP
AND       M02042
OUT       D002060.5	// L_1st BD Z JOG+
; L209
LOAD      D001060.0	// L_1st BD Z CTRL RDY
AND NOT   D001060.A	// L_1st BD Z WARNING
AND NOT   D001060.C	// L_1st BD Z SVD ERR
AND NOT   M02043
AND NOT   M00600	// EMERGENCY ALARM
OUT       D002060.1	// L_1st BD Z SERVO ON
; L210
LOAD      M0304C	// -
OUT       D002060.4	// L_1st BD Z HOME->
; L211
LOAD NOT  M03040
AND NOT   M01545
NOT
DMOV      D003400 D002072	// L_1st BD Z °¡¼Ó
DMOV      D003420 D002074	// L_1st BD Z °¨¼Ó
DMOV      D003440 D002062	// L_1st BD Z UP POS / L_1st BD Z ¸ñÇ¥À§Ä¡
DMOV      D003460 D002064	// L_1st BD Z ¸ñÇ¥¼Óµµ
AND       M01545
DMOV      1000 D002064	// L_1st BD Z ¸ñÇ¥¼Óµµ

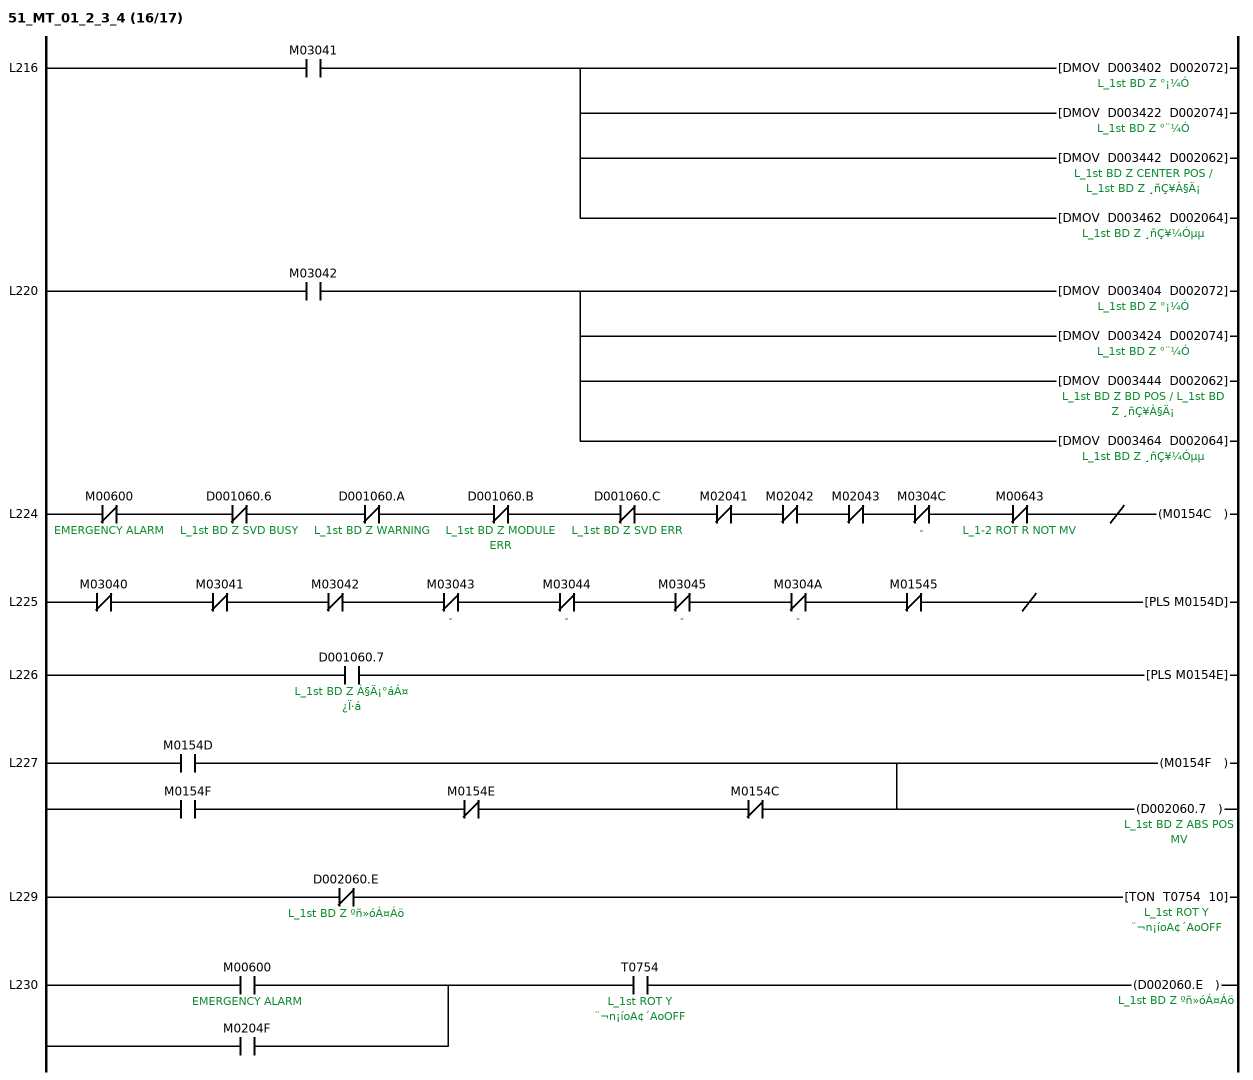
; L216
LOAD      M03041
DMOV      D003402 D002072	// L_1st BD Z °¡¼Ó
DMOV      D003422 D002074	// L_1st BD Z °¨¼Ó
DMOV      D003442 D002062	// L_1st BD Z CENTER POS / L_1st BD Z ¸ñÇ¥À§Ä¡
DMOV      D003462 D002064	// L_1st BD Z ¸ñÇ¥¼Óµµ
; L220
LOAD      M03042
DMOV      D003404 D002072	// L_1st BD Z °¡¼Ó
DMOV      D003424 D002074	// L_1st BD Z °¨¼Ó
DMOV      D003444 D002062	// L_1st BD Z BD POS / L_1st BD Z ¸ñÇ¥À§Ä¡
DMOV      D003464 D002064	// L_1st BD Z ¸ñÇ¥¼Óµµ
; L224
LOAD NOT  M00600	// EMERGENCY ALARM
AND NOT   D001060.6	// L_1st BD Z SVD BUSY
AND NOT   D001060.A	// L_1st BD Z WARNING
AND NOT   D001060.B	// L_1st BD Z MODULE ERR
AND NOT   D001060.C	// L_1st BD Z SVD ERR
AND NOT   M02041
AND NOT   M02042
AND NOT   M02043
AND NOT   M0304C	// -
AND NOT   M00643	// L_1-2 ROT R NOT MV
NOT
OUT       M0154C
; L225
LOAD NOT  M03040
AND NOT   M03041
AND NOT   M03042
AND NOT   M03043	// -
AND NOT   M03044	// -
AND NOT   M03045	// -
AND NOT   M0304A	// -
AND NOT   M01545
NOT
OUTP      M0154D
; L226
LOAD      D001060.7	// L_1st BD Z À§Ä¡°áÁ¤ ¿Ï·á
OUTP      M0154E
; L227
LOAD      M0154D
LOAD      M0154F
AND NOT   M0154E
AND NOT   M0154C
OR LOAD
OUT       M0154F
OUT       D002060.7	// L_1st BD Z ABS POS MV
; L229
LOAD NOT  D002060.E	// L_1st BD Z ºñ»óÁ¤Áö
TON       T0754 10	// L_1st ROT Y ¨¬n¡íoA¢´AoOFF
; L230
LOAD      M00600	// EMERGENCY ALARM
OR        M0204F
AND       T0754	// L_1st ROT Y ¨¬n¡íoA¢´AoOFF
OUT       D002060.E	// L_1st BD Z ºñ»óÁ¤Áö

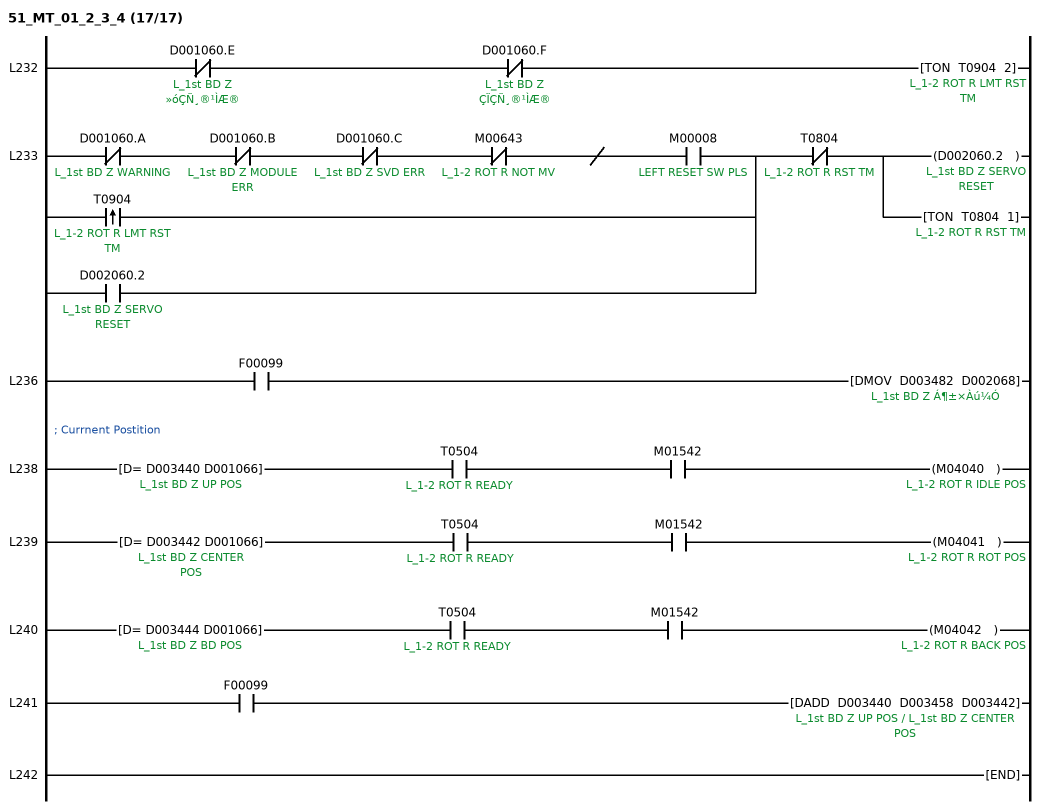
; L232
LOAD NOT  D001060.E	// L_1st BD Z »óÇÑ¸®¹ÌÆ®
AND NOT   D001060.F	// L_1st BD Z ÇÏÇÑ¸®¹ÌÆ®
TON       T0904 2	// L_1-2 ROT R LMT RST TM
; L233
LOAD NOT  D001060.A	// L_1st BD Z WARNING
AND NOT   D001060.B	// L_1st BD Z MODULE ERR
AND NOT   D001060.C	// L_1st BD Z SVD ERR
AND NOT   M00643	// L_1-2 ROT R NOT MV
NOT
AND       M00008	// LEFT RESET SW PLS
ORP       T0904	// L_1-2 ROT R LMT RST TM
OR        D002060.2	// L_1st BD Z SERVO RESET
AND NOT   T0804	// L_1-2 ROT R RST TM
OUT       D002060.2	// L_1st BD Z SERVO RESET
TON       T0804 1	// L_1-2 ROT R RST TM
; L236
LOAD      F00099
DMOV      D003482 D002068	// L_1st BD Z Á¶±×Àú¼Ó
// Currnent Postition
; L238
LOADD=    D003440 D001066	// L_1st BD Z UP POS
AND       T0504	// L_1-2 ROT R READY
AND       M01542
OUT       M04040	// L_1-2 ROT R IDLE POS
; L239
LOADD=    D003442 D001066	// L_1st BD Z CENTER POS
AND       T0504	// L_1-2 ROT R READY
AND       M01542
OUT       M04041	// L_1-2 ROT R ROT POS
; L240
LOADD=    D003444 D001066	// L_1st BD Z BD POS
AND       T0504	// L_1-2 ROT R READY
AND       M01542
OUT       M04042	// L_1-2 ROT R BACK POS
; L241
LOAD      F00099
DADD      D003440 D003458 D003442	// L_1st BD Z UP POS / L_1st BD Z CENTER POS
; L242
END

PROGRAM 52_MT_05_6_7_8 (task: ½ºÄµ ÇÁ·Î±×·¥)

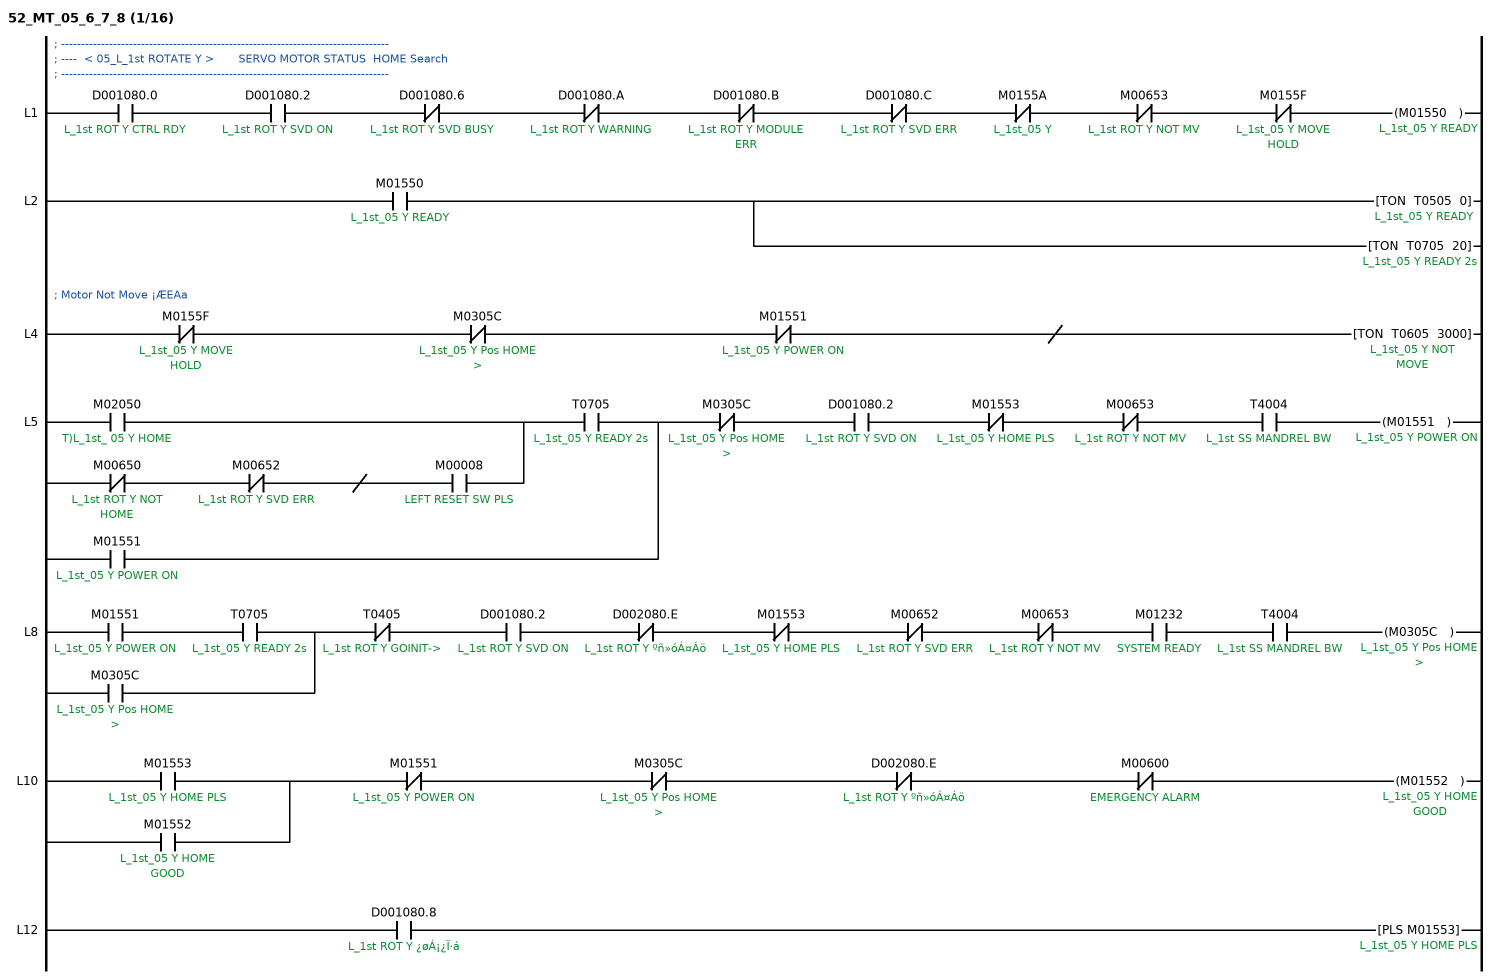
// ----------------------------------------------------------------------------------
// 
// ----  < 05_L_1st ROTATE Y >       SERVO MOTOR STATUS  HOME Search
// 
// ----------------------------------------------------------------------------------
; L1
LOAD      D001080.0	// L_1st ROT Y CTRL RDY
AND       D001080.2	// L_1st ROT Y SVD ON
AND NOT   D001080.6	// L_1st ROT Y SVD BUSY
AND NOT   D001080.A	// L_1st ROT Y WARNING
AND NOT   D001080.B	// L_1st ROT Y MODULE ERR
AND NOT   D001080.C	// L_1st ROT Y SVD ERR
AND NOT   M0155A	// L_1st_05 Y
AND NOT   M00653	// L_1st ROT Y NOT MV
AND NOT   M0155F	// L_1st_05 Y MOVE HOLD
OUT       M01550	// L_1st_05 Y READY
; L2
LOAD      M01550	// L_1st_05 Y READY
TON       T0505 0	// L_1st_05 Y READY
TON       T0705 20	// L_1st_05 Y READY 2s
; L4
LOAD NOT  M0155F	// L_1st_05 Y MOVE HOLD
AND NOT   M0305C	// L_1st_05 Y Pos HOME >
AND NOT   M01551	// L_1st_05 Y POWER ON
NOT
TON       T0605 3000	// L_1st_05 Y NOT MOVE
// output comment: Motor Not Move ¡ÆEAa
; L5
LOAD      M02050	// T)L_1st_ 05 Y HOME
LOAD NOT  M00650	// L_1st ROT Y NOT HOME
AND NOT   M00652	// L_1st ROT Y SVD ERR
NOT
AND       M00008	// LEFT RESET SW PLS
OR LOAD
AND       T0705	// L_1st_05 Y READY 2s
OR        M01551	// L_1st_05 Y POWER ON
AND NOT   M0305C	// L_1st_05 Y Pos HOME >
AND       D001080.2	// L_1st ROT Y SVD ON
AND NOT   M01553	// L_1st_05 Y HOME PLS
AND NOT   M00653	// L_1st ROT Y NOT MV
AND       T4004	// L_1st SS MANDREL BW
OUT       M01551	// L_1st_05 Y POWER ON
; L8
LOAD      M01551	// L_1st_05 Y POWER ON
AND       T0705	// L_1st_05 Y READY 2s
OR        M0305C	// L_1st_05 Y Pos HOME >
AND NOT   T0405	// L_1st ROT Y GOINIT->
AND       D001080.2	// L_1st ROT Y SVD ON
AND NOT   D002080.E	// L_1st ROT Y ºñ»óÁ¤Áö
AND NOT   M01553	// L_1st_05 Y HOME PLS
AND NOT   M00652	// L_1st ROT Y SVD ERR
AND NOT   M00653	// L_1st ROT Y NOT MV
AND       M01232	// SYSTEM READY
AND       T4004	// L_1st SS MANDREL BW
OUT       M0305C	// L_1st_05 Y Pos HOME >
; L10
LOAD      M01553	// L_1st_05 Y HOME PLS
OR        M01552	// L_1st_05 Y HOME GOOD
AND NOT   M01551	// L_1st_05 Y POWER ON
AND NOT   M0305C	// L_1st_05 Y Pos HOME >
AND NOT   D002080.E	// L_1st ROT Y ºñ»óÁ¤Áö
AND NOT   M00600	// EMERGENCY ALARM
OUT       M01552	// L_1st_05 Y HOME GOOD
; L12
LOAD      D001080.8	// L_1st ROT Y ¿øÁ¡¿Ï·á
OUTP      M01553	// L_1st_05 Y HOME PLS

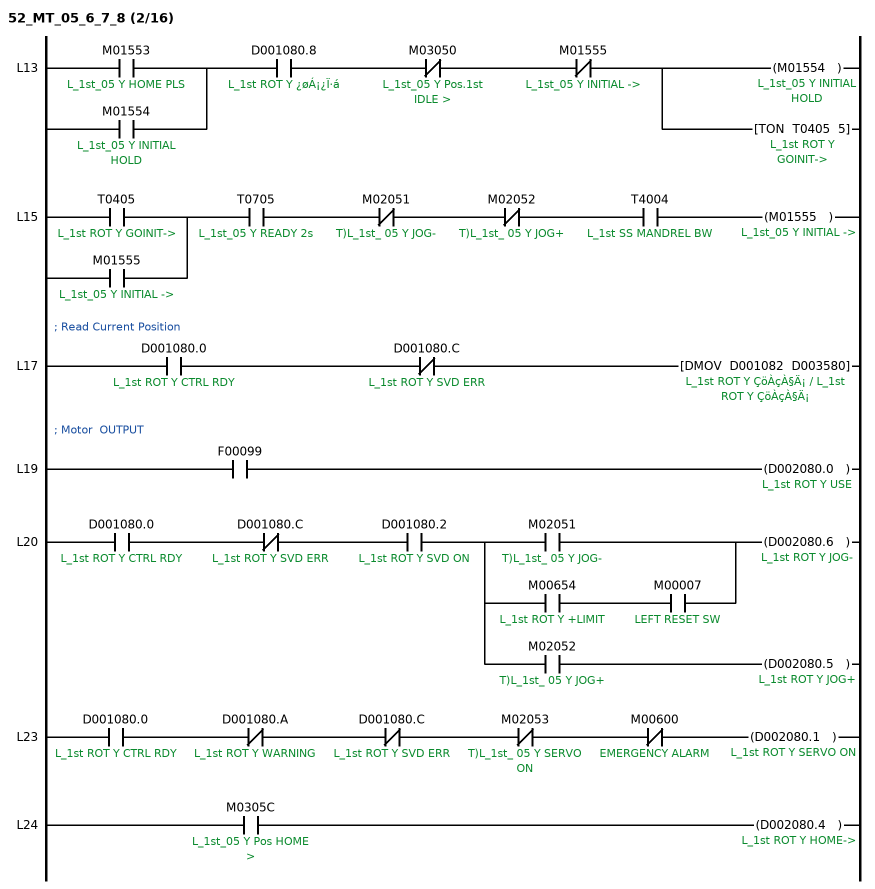
; L13
LOAD      M01553	// L_1st_05 Y HOME PLS
OR        M01554	// L_1st_05 Y INITIAL HOLD
AND       D001080.8	// L_1st ROT Y ¿øÁ¡¿Ï·á
AND NOT   M03050	// L_1st_05 Y Pos.1st IDLE >
AND NOT   M01555	// L_1st_05 Y INITIAL ->
OUT       M01554	// L_1st_05 Y INITIAL HOLD
TON       T0405 5	// L_1st ROT Y GOINIT->
; L15
LOAD      T0405	// L_1st ROT Y GOINIT->
OR        M01555	// L_1st_05 Y INITIAL ->
AND       T0705	// L_1st_05 Y READY 2s
AND NOT   M02051	// T)L_1st_ 05 Y JOG-
AND NOT   M02052	// T)L_1st_ 05 Y JOG+
AND       T4004	// L_1st SS MANDREL BW
OUT       M01555	// L_1st_05 Y INITIAL ->
; L17
LOAD      D001080.0	// L_1st ROT Y CTRL RDY
AND NOT   D001080.C	// L_1st ROT Y SVD ERR
DMOV      D001082 D003580	// L_1st ROT Y ÇöÀçÀ§Ä¡ / L_1st ROT Y ÇöÀçÀ§Ä¡
// output comment: Read Current Position
//  Motor  OUTPUT
; L19
LOAD      F00099
OUT       D002080.0	// L_1st ROT Y USE
; L20
LOAD      D001080.0	// L_1st ROT Y CTRL RDY
AND NOT   D001080.C	// L_1st ROT Y SVD ERR
AND       D001080.2	// L_1st ROT Y SVD ON
MPUSH
LOAD      M02051	// T)L_1st_ 05 Y JOG-
LOAD      M00654	// L_1st ROT Y +LIMIT
AND       M00007	// LEFT RESET SW
OR LOAD
AND LOAD
OUT       D002080.6	// L_1st ROT Y JOG-
MPOP
AND       M02052	// T)L_1st_ 05 Y JOG+
OUT       D002080.5	// L_1st ROT Y JOG+
; L23
LOAD      D001080.0	// L_1st ROT Y CTRL RDY
AND NOT   D001080.A	// L_1st ROT Y WARNING
AND NOT   D001080.C	// L_1st ROT Y SVD ERR
AND NOT   M02053	// T)L_1st_ 05 Y SERVO ON
AND NOT   M00600	// EMERGENCY ALARM
OUT       D002080.1	// L_1st ROT Y SERVO ON
; L24
LOAD      M0305C	// L_1st_05 Y Pos HOME >
OUT       D002080.4	// L_1st ROT Y HOME->

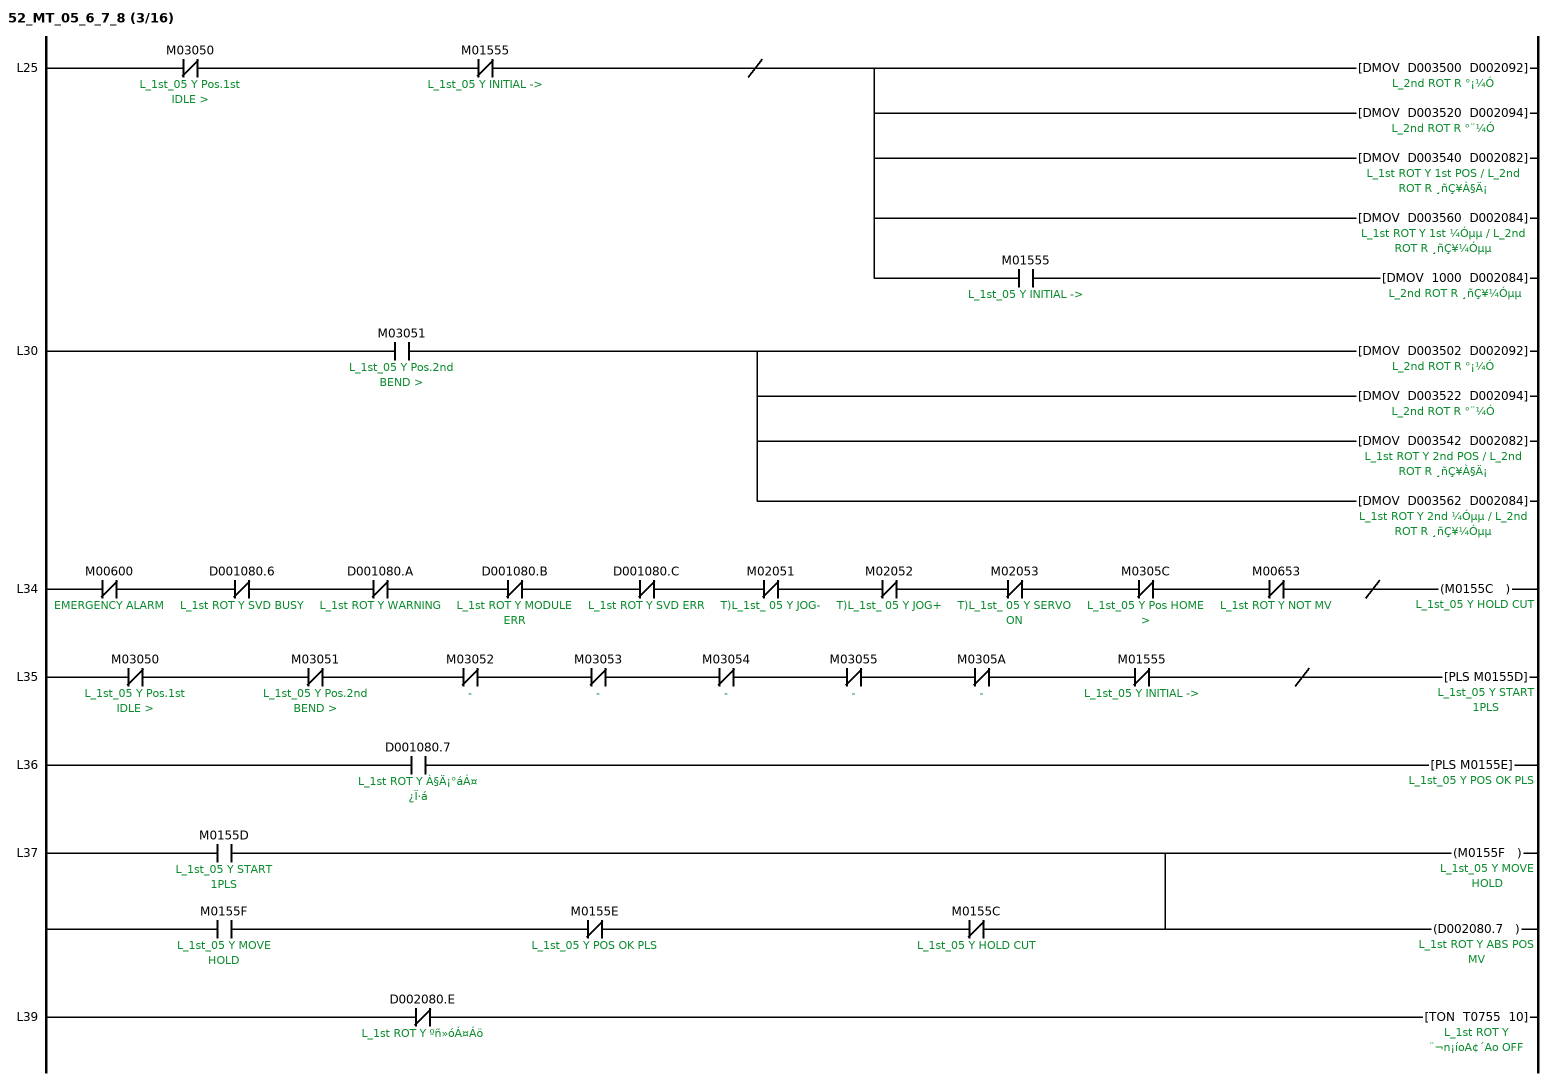
; L25
LOAD NOT  M03050	// L_1st_05 Y Pos.1st IDLE >
AND NOT   M01555	// L_1st_05 Y INITIAL ->
NOT
DMOV      D003500 D002092	// L_2nd ROT R °¡¼Ó
DMOV      D003520 D002094	// L_2nd ROT R °¨¼Ó
DMOV      D003540 D002082	// L_1st ROT Y 1st POS / L_2nd ROT R ¸ñÇ¥À§Ä¡
DMOV      D003560 D002084	// L_1st ROT Y 1st ¼Óµµ / L_2nd ROT R ¸ñÇ¥¼Óµµ
AND       M01555	// L_1st_05 Y INITIAL ->
DMOV      1000 D002084	// L_2nd ROT R ¸ñÇ¥¼Óµµ
; L30
LOAD      M03051	// L_1st_05 Y Pos.2nd BEND >
DMOV      D003502 D002092	// L_2nd ROT R °¡¼Ó
DMOV      D003522 D002094	// L_2nd ROT R °¨¼Ó
DMOV      D003542 D002082	// L_1st ROT Y 2nd POS / L_2nd ROT R ¸ñÇ¥À§Ä¡
DMOV      D003562 D002084	// L_1st ROT Y 2nd ¼Óµµ / L_2nd ROT R ¸ñÇ¥¼Óµµ
; L34
LOAD NOT  M00600	// EMERGENCY ALARM
AND NOT   D001080.6	// L_1st ROT Y SVD BUSY
AND NOT   D001080.A	// L_1st ROT Y WARNING
AND NOT   D001080.B	// L_1st ROT Y MODULE ERR
AND NOT   D001080.C	// L_1st ROT Y SVD ERR
AND NOT   M02051	// T)L_1st_ 05 Y JOG-
AND NOT   M02052	// T)L_1st_ 05 Y JOG+
AND NOT   M02053	// T)L_1st_ 05 Y SERVO ON
AND NOT   M0305C	// L_1st_05 Y Pos HOME >
AND NOT   M00653	// L_1st ROT Y NOT MV
NOT
OUT       M0155C	// L_1st_05 Y HOLD CUT
; L35
LOAD NOT  M03050	// L_1st_05 Y Pos.1st IDLE >
AND NOT   M03051	// L_1st_05 Y Pos.2nd BEND >
AND NOT   M03052	// -
AND NOT   M03053	// -
AND NOT   M03054	// -
AND NOT   M03055	// -
AND NOT   M0305A	// -
AND NOT   M01555	// L_1st_05 Y INITIAL ->
NOT
OUTP      M0155D	// L_1st_05 Y START 1PLS
; L36
LOAD      D001080.7	// L_1st ROT Y À§Ä¡°áÁ¤ ¿Ï·á
OUTP      M0155E	// L_1st_05 Y POS OK PLS
; L37
LOAD      M0155D	// L_1st_05 Y START 1PLS
LOAD      M0155F	// L_1st_05 Y MOVE HOLD
AND NOT   M0155E	// L_1st_05 Y POS OK PLS
AND NOT   M0155C	// L_1st_05 Y HOLD CUT
OR LOAD
OUT       M0155F	// L_1st_05 Y MOVE HOLD
OUT       D002080.7	// L_1st ROT Y ABS POS MV
; L39
LOAD NOT  D002080.E	// L_1st ROT Y ºñ»óÁ¤Áö
TON       T0755 10	// L_1st ROT Y ¨¬n¡íoA¢´Ao OFF

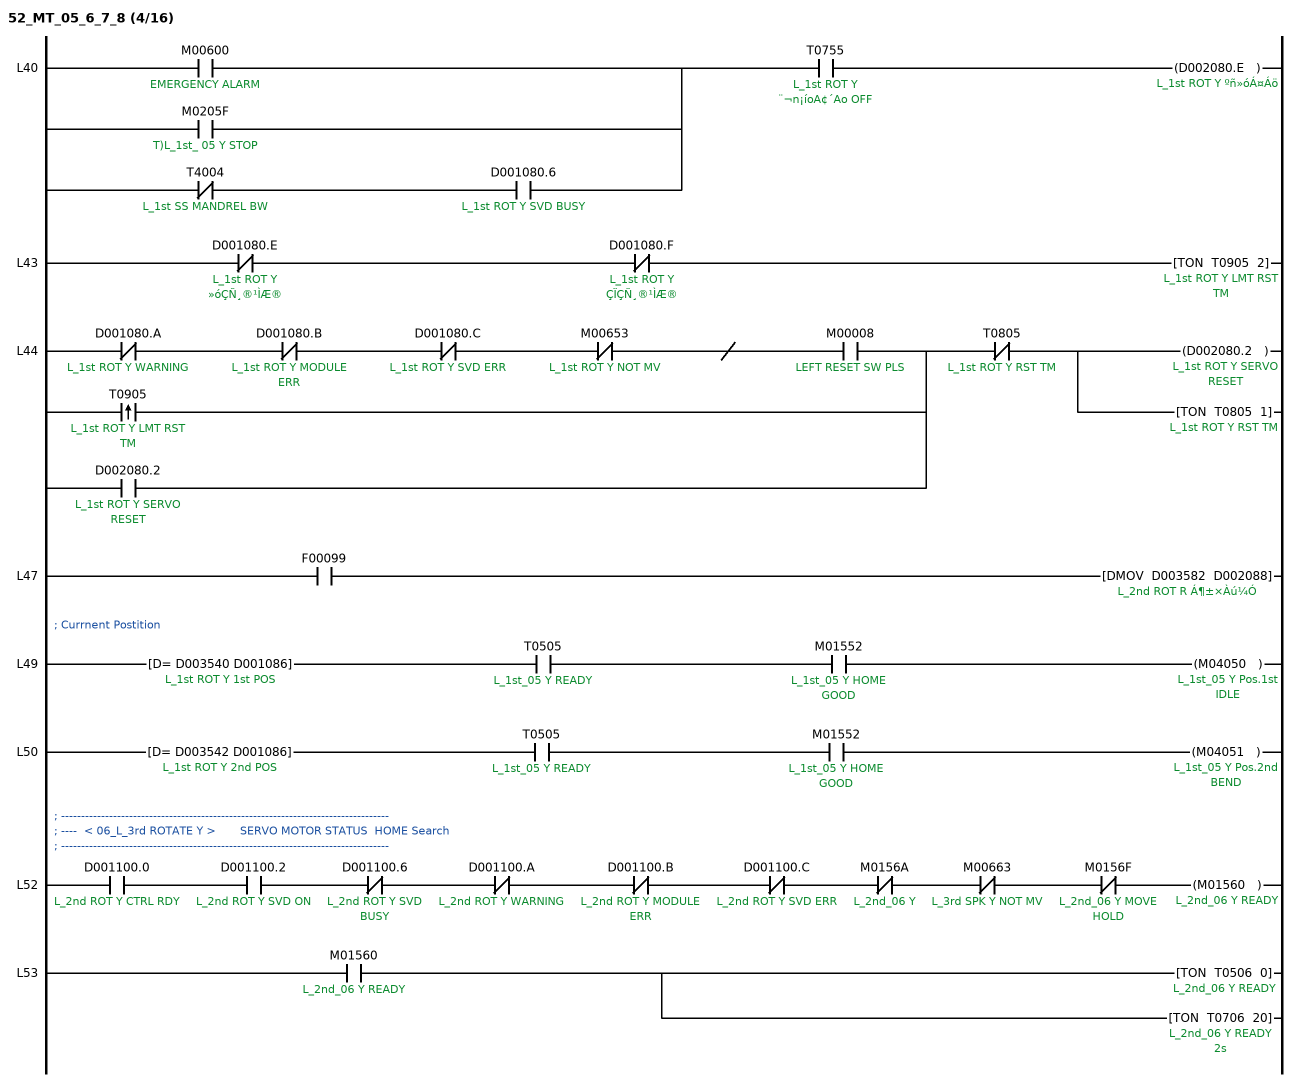
; L40
LOAD      M00600	// EMERGENCY ALARM
OR        M0205F	// T)L_1st_ 05 Y STOP
LOAD NOT  T4004	// L_1st SS MANDREL BW
AND       D001080.6	// L_1st ROT Y SVD BUSY
OR LOAD
AND       T0755	// L_1st ROT Y ¨¬n¡íoA¢´Ao OFF
OUT       D002080.E	// L_1st ROT Y ºñ»óÁ¤Áö
; L43
LOAD NOT  D001080.E	// L_1st ROT Y »óÇÑ¸®¹ÌÆ®
AND NOT   D001080.F	// L_1st ROT Y ÇÏÇÑ¸®¹ÌÆ®
TON       T0905 2	// L_1st ROT Y LMT RST TM
; L44
LOAD NOT  D001080.A	// L_1st ROT Y WARNING
AND NOT   D001080.B	// L_1st ROT Y MODULE ERR
AND NOT   D001080.C	// L_1st ROT Y SVD ERR
AND NOT   M00653	// L_1st ROT Y NOT MV
NOT
AND       M00008	// LEFT RESET SW PLS
ORP       T0905	// L_1st ROT Y LMT RST TM
OR        D002080.2	// L_1st ROT Y SERVO RESET
AND NOT   T0805	// L_1st ROT Y RST TM
OUT       D002080.2	// L_1st ROT Y SERVO RESET
TON       T0805 1	// L_1st ROT Y RST TM
; L47
LOAD      F00099
DMOV      D003582 D002088	// L_2nd ROT R Á¶±×Àú¼Ó
// Currnent Postition
; L49
LOADD=    D003540 D001086	// L_1st ROT Y 1st POS
AND       T0505	// L_1st_05 Y READY
AND       M01552	// L_1st_05 Y HOME GOOD
OUT       M04050	// L_1st_05 Y Pos.1st IDLE
; L50
LOADD=    D003542 D001086	// L_1st ROT Y 2nd POS
AND       T0505	// L_1st_05 Y READY
AND       M01552	// L_1st_05 Y HOME GOOD
OUT       M04051	// L_1st_05 Y Pos.2nd BEND
// ----------------------------------------------------------------------------------
// 
// ----  < 06_L_3rd ROTATE Y >       SERVO MOTOR STATUS  HOME Search
// 
// ----------------------------------------------------------------------------------
; L52
LOAD      D001100.0	// L_2nd ROT Y CTRL RDY
AND       D001100.2	// L_2nd ROT Y SVD ON
AND NOT   D001100.6	// L_2nd ROT Y SVD BUSY
AND NOT   D001100.A	// L_2nd ROT Y WARNING
AND NOT   D001100.B	// L_2nd ROT Y MODULE ERR
AND NOT   D001100.C	// L_2nd ROT Y SVD ERR
AND NOT   M0156A	// L_2nd_06 Y
AND NOT   M00663	// L_3rd SPK Y NOT MV
AND NOT   M0156F	// L_2nd_06 Y MOVE HOLD
OUT       M01560	// L_2nd_06 Y READY
; L53
LOAD      M01560	// L_2nd_06 Y READY
TON       T0506 0	// L_2nd_06 Y READY
TON       T0706 20	// L_2nd_06 Y READY 2s

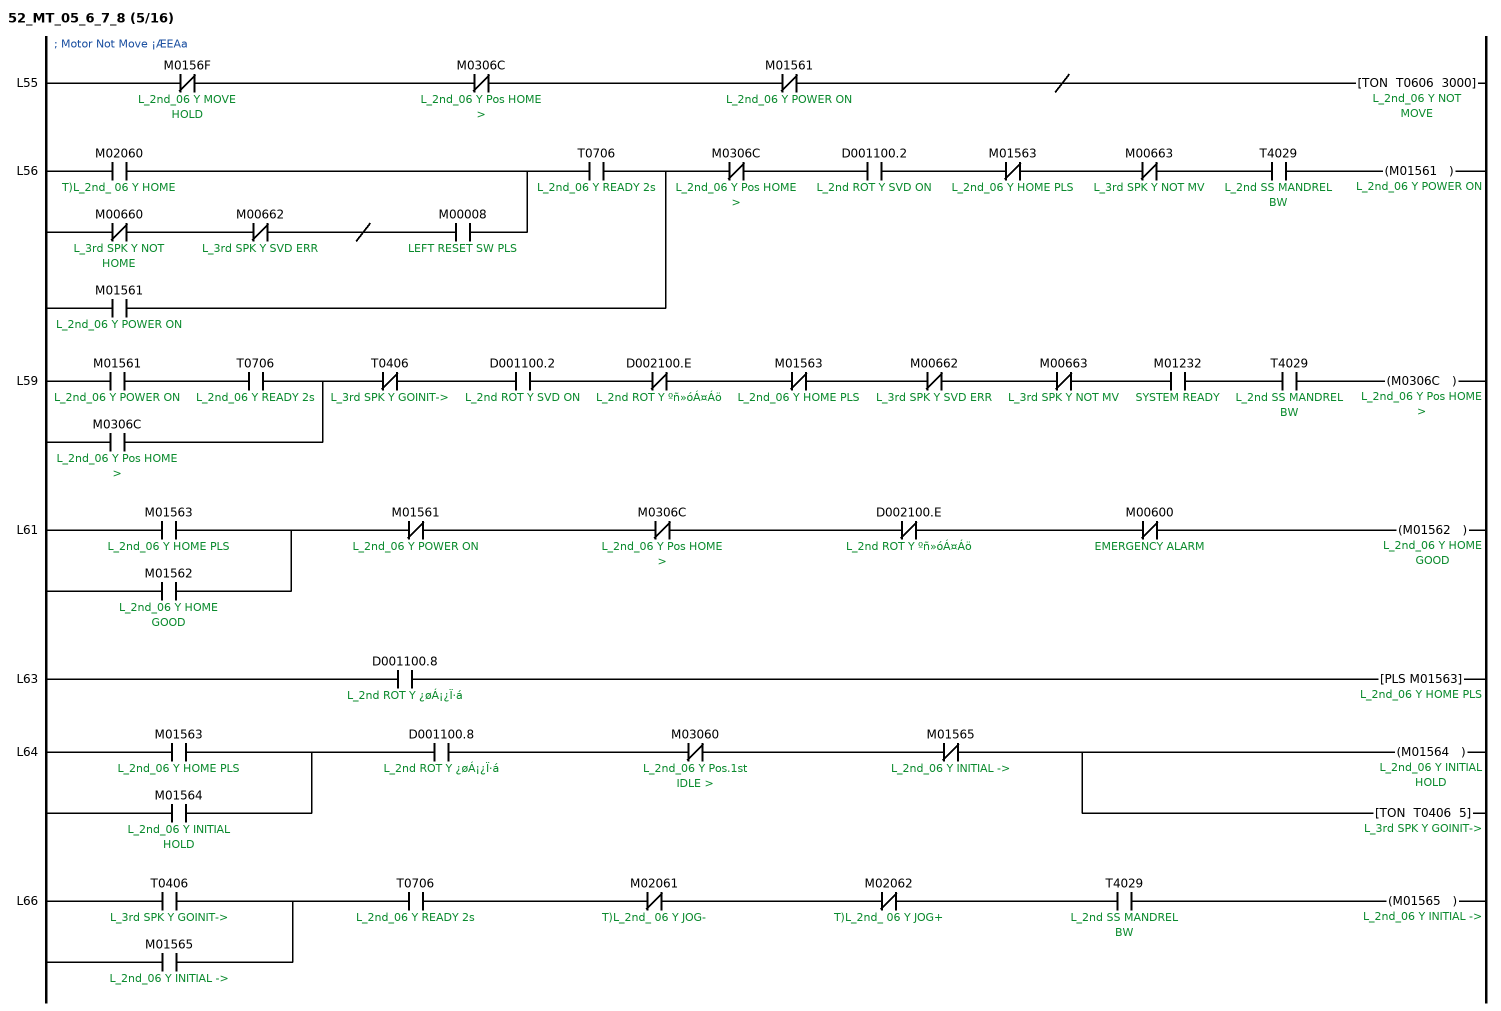
; L55
LOAD NOT  M0156F	// L_2nd_06 Y MOVE HOLD
AND NOT   M0306C	// L_2nd_06 Y Pos HOME >
AND NOT   M01561	// L_2nd_06 Y POWER ON
NOT
TON       T0606 3000	// L_2nd_06 Y NOT MOVE
// output comment: Motor Not Move ¡ÆEAa
; L56
LOAD      M02060	// T)L_2nd_ 06 Y HOME
LOAD NOT  M00660	// L_3rd SPK Y NOT HOME
AND NOT   M00662	// L_3rd SPK Y SVD ERR
NOT
AND       M00008	// LEFT RESET SW PLS
OR LOAD
AND       T0706	// L_2nd_06 Y READY 2s
OR        M01561	// L_2nd_06 Y POWER ON
AND NOT   M0306C	// L_2nd_06 Y Pos HOME >
AND       D001100.2	// L_2nd ROT Y SVD ON
AND NOT   M01563	// L_2nd_06 Y HOME PLS
AND NOT   M00663	// L_3rd SPK Y NOT MV
AND       T4029	// L_2nd SS MANDREL BW
OUT       M01561	// L_2nd_06 Y POWER ON
; L59
LOAD      M01561	// L_2nd_06 Y POWER ON
AND       T0706	// L_2nd_06 Y READY 2s
OR        M0306C	// L_2nd_06 Y Pos HOME >
AND NOT   T0406	// L_3rd SPK Y GOINIT->
AND       D001100.2	// L_2nd ROT Y SVD ON
AND NOT   D002100.E	// L_2nd ROT Y ºñ»óÁ¤Áö
AND NOT   M01563	// L_2nd_06 Y HOME PLS
AND NOT   M00662	// L_3rd SPK Y SVD ERR
AND NOT   M00663	// L_3rd SPK Y NOT MV
AND       M01232	// SYSTEM READY
AND       T4029	// L_2nd SS MANDREL BW
OUT       M0306C	// L_2nd_06 Y Pos HOME >
; L61
LOAD      M01563	// L_2nd_06 Y HOME PLS
OR        M01562	// L_2nd_06 Y HOME GOOD
AND NOT   M01561	// L_2nd_06 Y POWER ON
AND NOT   M0306C	// L_2nd_06 Y Pos HOME >
AND NOT   D002100.E	// L_2nd ROT Y ºñ»óÁ¤Áö
AND NOT   M00600	// EMERGENCY ALARM
OUT       M01562	// L_2nd_06 Y HOME GOOD
; L63
LOAD      D001100.8	// L_2nd ROT Y ¿øÁ¡¿Ï·á
OUTP      M01563	// L_2nd_06 Y HOME PLS
; L64
LOAD      M01563	// L_2nd_06 Y HOME PLS
OR        M01564	// L_2nd_06 Y INITIAL HOLD
AND       D001100.8	// L_2nd ROT Y ¿øÁ¡¿Ï·á
AND NOT   M03060	// L_2nd_06 Y Pos.1st IDLE >
AND NOT   M01565	// L_2nd_06 Y INITIAL ->
OUT       M01564	// L_2nd_06 Y INITIAL HOLD
TON       T0406 5	// L_3rd SPK Y GOINIT->
; L66
LOAD      T0406	// L_3rd SPK Y GOINIT->
OR        M01565	// L_2nd_06 Y INITIAL ->
AND       T0706	// L_2nd_06 Y READY 2s
AND NOT   M02061	// T)L_2nd_ 06 Y JOG-
AND NOT   M02062	// T)L_2nd_ 06 Y JOG+
AND       T4029	// L_2nd SS MANDREL BW
OUT       M01565	// L_2nd_06 Y INITIAL ->

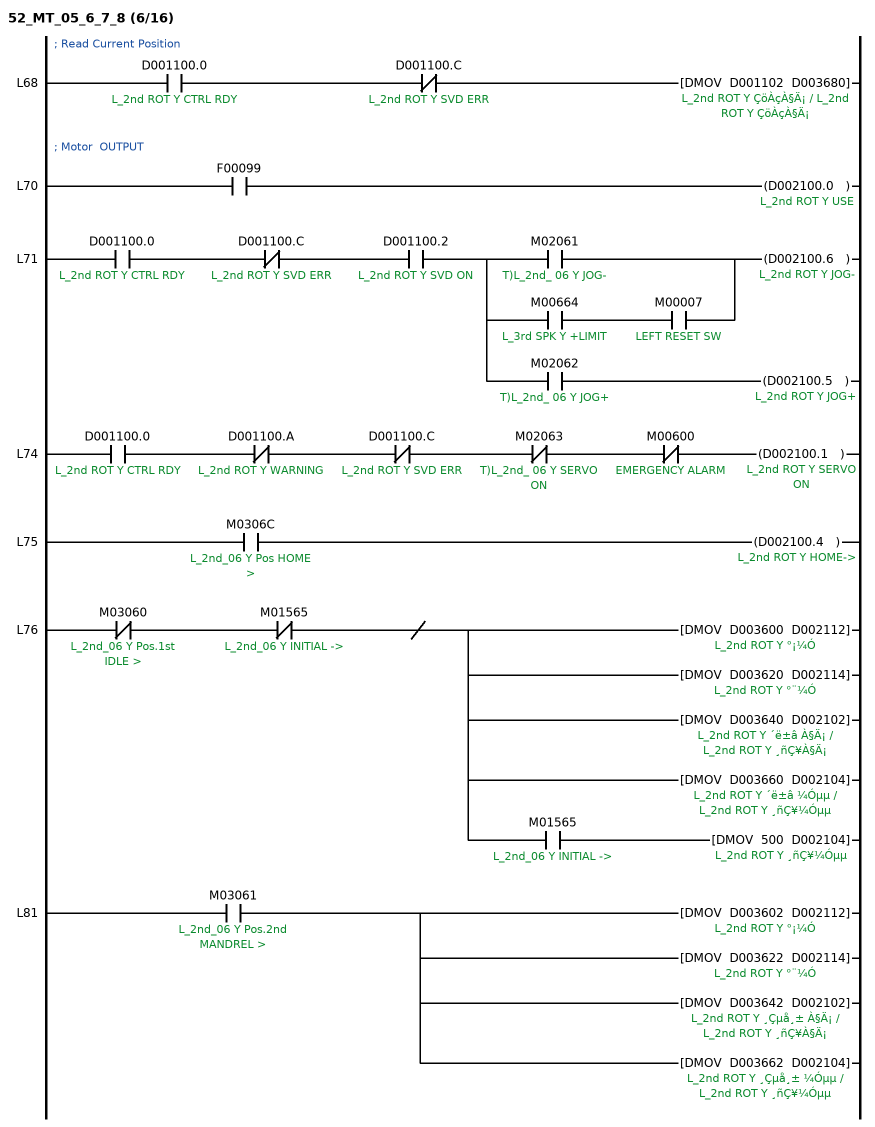
; L68
LOAD      D001100.0	// L_2nd ROT Y CTRL RDY
AND NOT   D001100.C	// L_2nd ROT Y SVD ERR
DMOV      D001102 D003680	// L_2nd ROT Y ÇöÀçÀ§Ä¡ / L_2nd ROT Y ÇöÀçÀ§Ä¡
// output comment: Read Current Position
//  Motor  OUTPUT
; L70
LOAD      F00099
OUT       D002100.0	// L_2nd ROT Y USE
; L71
LOAD      D001100.0	// L_2nd ROT Y CTRL RDY
AND NOT   D001100.C	// L_2nd ROT Y SVD ERR
AND       D001100.2	// L_2nd ROT Y SVD ON
MPUSH
LOAD      M02061	// T)L_2nd_ 06 Y JOG-
LOAD      M00664	// L_3rd SPK Y +LIMIT
AND       M00007	// LEFT RESET SW
OR LOAD
AND LOAD
OUT       D002100.6	// L_2nd ROT Y JOG-
MPOP
AND       M02062	// T)L_2nd_ 06 Y JOG+
OUT       D002100.5	// L_2nd ROT Y JOG+
; L74
LOAD      D001100.0	// L_2nd ROT Y CTRL RDY
AND NOT   D001100.A	// L_2nd ROT Y WARNING
AND NOT   D001100.C	// L_2nd ROT Y SVD ERR
AND NOT   M02063	// T)L_2nd_ 06 Y SERVO ON
AND NOT   M00600	// EMERGENCY ALARM
OUT       D002100.1	// L_2nd ROT Y SERVO ON
; L75
LOAD      M0306C	// L_2nd_06 Y Pos HOME >
OUT       D002100.4	// L_2nd ROT Y HOME->
; L76
LOAD NOT  M03060	// L_2nd_06 Y Pos.1st IDLE >
AND NOT   M01565	// L_2nd_06 Y INITIAL ->
NOT
DMOV      D003600 D002112	// L_2nd ROT Y °¡¼Ó
DMOV      D003620 D002114	// L_2nd ROT Y °¨¼Ó
DMOV      D003640 D002102	// L_2nd ROT Y ´ë±â À§Ä¡ / L_2nd ROT Y ¸ñÇ¥À§Ä¡
DMOV      D003660 D002104	// L_2nd ROT Y ´ë±â ¼Óµµ / L_2nd ROT Y ¸ñÇ¥¼Óµµ
AND       M01565	// L_2nd_06 Y INITIAL ->
DMOV      500 D002104	// L_2nd ROT Y ¸ñÇ¥¼Óµµ
; L81
LOAD      M03061	// L_2nd_06 Y Pos.2nd MANDREL >
DMOV      D003602 D002112	// L_2nd ROT Y °¡¼Ó
DMOV      D003622 D002114	// L_2nd ROT Y °¨¼Ó
DMOV      D003642 D002102	// L_2nd ROT Y ¸Çµå¸± À§Ä¡ / L_2nd ROT Y ¸ñÇ¥À§Ä¡
DMOV      D003662 D002104	// L_2nd ROT Y ¸Çµå¸± ¼Óµµ / L_2nd ROT Y ¸ñÇ¥¼Óµµ

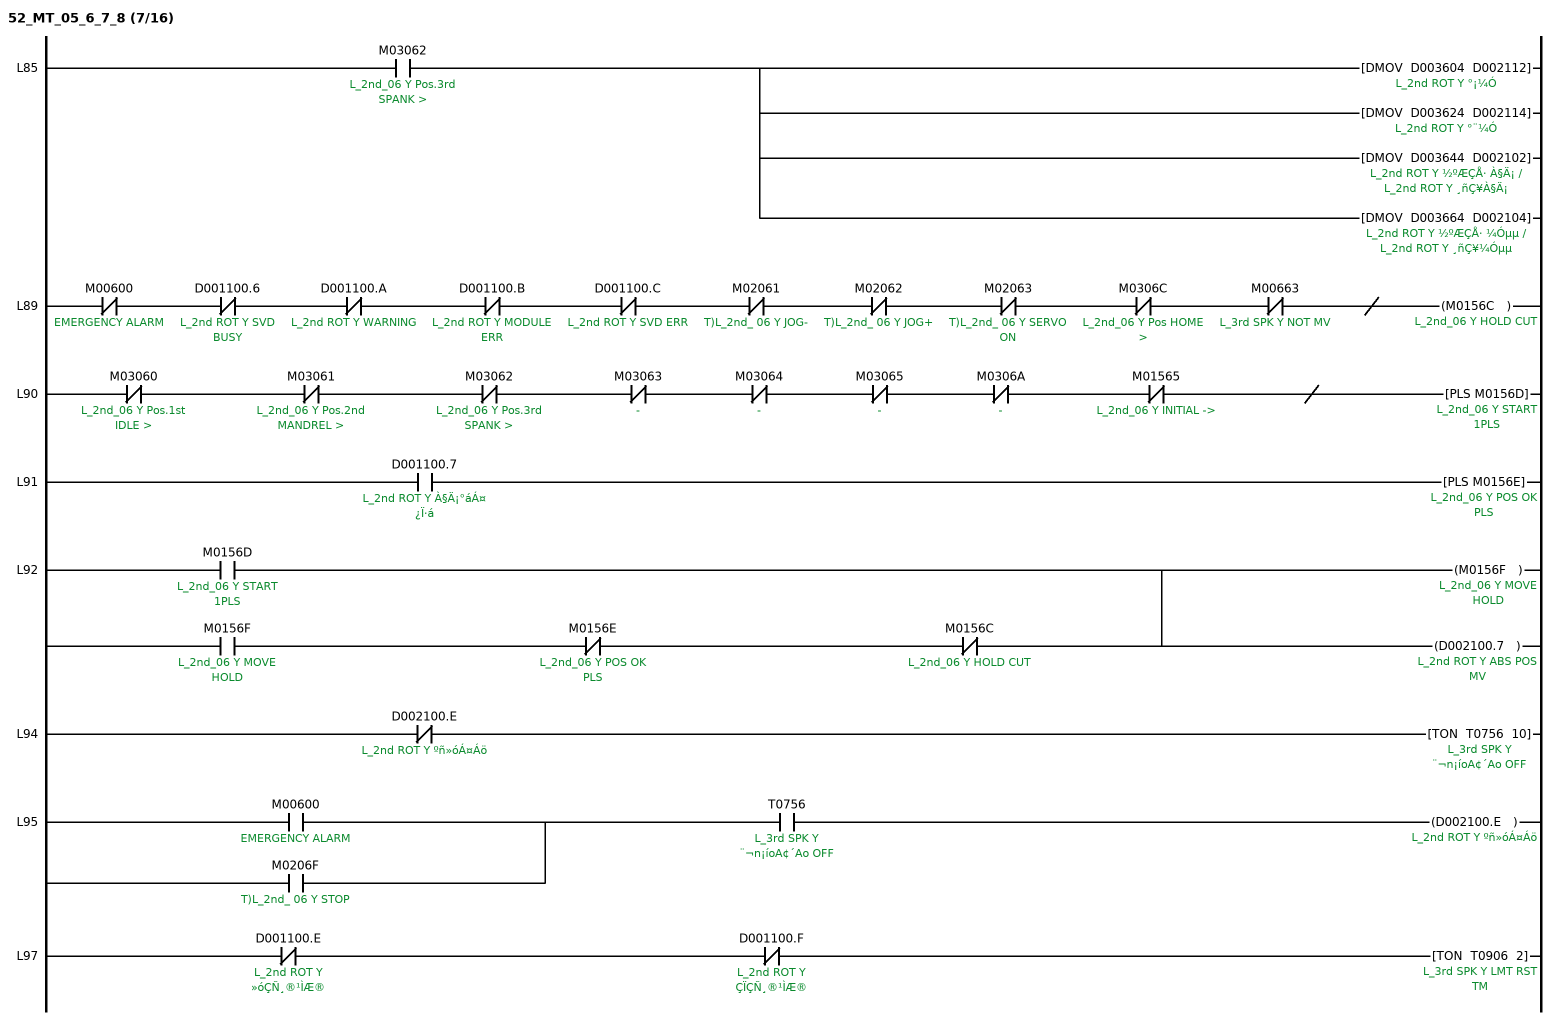
; L85
LOAD      M03062	// L_2nd_06 Y Pos.3rd SPANK >
DMOV      D003604 D002112	// L_2nd ROT Y °¡¼Ó
DMOV      D003624 D002114	// L_2nd ROT Y °¨¼Ó
DMOV      D003644 D002102	// L_2nd ROT Y ½ºÆÇÅ· À§Ä¡ / L_2nd ROT Y ¸ñÇ¥À§Ä¡
DMOV      D003664 D002104	// L_2nd ROT Y ½ºÆÇÅ· ¼Óµµ / L_2nd ROT Y ¸ñÇ¥¼Óµµ
; L89
LOAD NOT  M00600	// EMERGENCY ALARM
AND NOT   D001100.6	// L_2nd ROT Y SVD BUSY
AND NOT   D001100.A	// L_2nd ROT Y WARNING
AND NOT   D001100.B	// L_2nd ROT Y MODULE ERR
AND NOT   D001100.C	// L_2nd ROT Y SVD ERR
AND NOT   M02061	// T)L_2nd_ 06 Y JOG-
AND NOT   M02062	// T)L_2nd_ 06 Y JOG+
AND NOT   M02063	// T)L_2nd_ 06 Y SERVO ON
AND NOT   M0306C	// L_2nd_06 Y Pos HOME >
AND NOT   M00663	// L_3rd SPK Y NOT MV
NOT
OUT       M0156C	// L_2nd_06 Y HOLD CUT
; L90
LOAD NOT  M03060	// L_2nd_06 Y Pos.1st IDLE >
AND NOT   M03061	// L_2nd_06 Y Pos.2nd MANDREL >
AND NOT   M03062	// L_2nd_06 Y Pos.3rd SPANK >
AND NOT   M03063	// -
AND NOT   M03064	// -
AND NOT   M03065	// -
AND NOT   M0306A	// -
AND NOT   M01565	// L_2nd_06 Y INITIAL ->
NOT
OUTP      M0156D	// L_2nd_06 Y START 1PLS
; L91
LOAD      D001100.7	// L_2nd ROT Y À§Ä¡°áÁ¤ ¿Ï·á
OUTP      M0156E	// L_2nd_06 Y POS OK PLS
; L92
LOAD      M0156D	// L_2nd_06 Y START 1PLS
LOAD      M0156F	// L_2nd_06 Y MOVE HOLD
AND NOT   M0156E	// L_2nd_06 Y POS OK PLS
AND NOT   M0156C	// L_2nd_06 Y HOLD CUT
OR LOAD
OUT       M0156F	// L_2nd_06 Y MOVE HOLD
OUT       D002100.7	// L_2nd ROT Y ABS POS MV
; L94
LOAD NOT  D002100.E	// L_2nd ROT Y ºñ»óÁ¤Áö
TON       T0756 10	// L_3rd SPK Y ¨¬n¡íoA¢´Ao OFF
; L95
LOAD      M00600	// EMERGENCY ALARM
OR        M0206F	// T)L_2nd_ 06 Y STOP
AND       T0756	// L_3rd SPK Y ¨¬n¡íoA¢´Ao OFF
OUT       D002100.E	// L_2nd ROT Y ºñ»óÁ¤Áö
; L97
LOAD NOT  D001100.E	// L_2nd ROT Y »óÇÑ¸®¹ÌÆ®
AND NOT   D001100.F	// L_2nd ROT Y ÇÏÇÑ¸®¹ÌÆ®
TON       T0906 2	// L_3rd SPK Y LMT RST TM

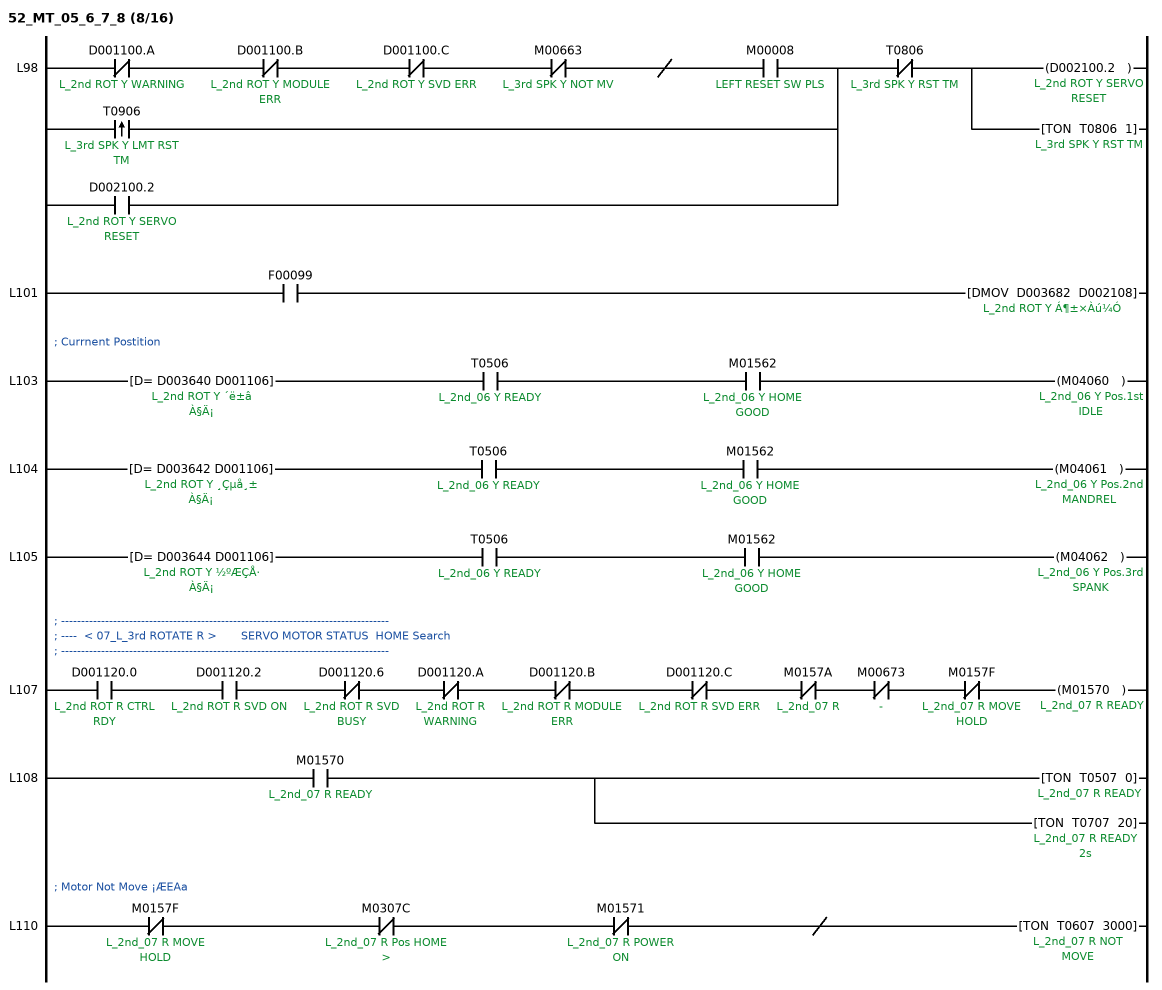
; L98
LOAD NOT  D001100.A	// L_2nd ROT Y WARNING
AND NOT   D001100.B	// L_2nd ROT Y MODULE ERR
AND NOT   D001100.C	// L_2nd ROT Y SVD ERR
AND NOT   M00663	// L_3rd SPK Y NOT MV
NOT
AND       M00008	// LEFT RESET SW PLS
ORP       T0906	// L_3rd SPK Y LMT RST TM
OR        D002100.2	// L_2nd ROT Y SERVO RESET
AND NOT   T0806	// L_3rd SPK Y RST TM
OUT       D002100.2	// L_2nd ROT Y SERVO RESET
TON       T0806 1	// L_3rd SPK Y RST TM
; L101
LOAD      F00099
DMOV      D003682 D002108	// L_2nd ROT Y Á¶±×Àú¼Ó
// Currnent Postition
; L103
LOADD=    D003640 D001106	// L_2nd ROT Y ´ë±â À§Ä¡
AND       T0506	// L_2nd_06 Y READY
AND       M01562	// L_2nd_06 Y HOME GOOD
OUT       M04060	// L_2nd_06 Y Pos.1st IDLE
; L104
LOADD=    D003642 D001106	// L_2nd ROT Y ¸Çµå¸± À§Ä¡
AND       T0506	// L_2nd_06 Y READY
AND       M01562	// L_2nd_06 Y HOME GOOD
OUT       M04061	// L_2nd_06 Y Pos.2nd MANDREL
; L105
LOADD=    D003644 D001106	// L_2nd ROT Y ½ºÆÇÅ· À§Ä¡
AND       T0506	// L_2nd_06 Y READY
AND       M01562	// L_2nd_06 Y HOME GOOD
OUT       M04062	// L_2nd_06 Y Pos.3rd SPANK
// ----------------------------------------------------------------------------------
// 
// ----  < 07_L_3rd ROTATE R >       SERVO MOTOR STATUS  HOME Search
// 
// ----------------------------------------------------------------------------------
; L107
LOAD      D001120.0	// L_2nd ROT R CTRL RDY
AND       D001120.2	// L_2nd ROT R SVD ON
AND NOT   D001120.6	// L_2nd ROT R SVD BUSY
AND NOT   D001120.A	// L_2nd ROT R WARNING
AND NOT   D001120.B	// L_2nd ROT R MODULE ERR
AND NOT   D001120.C	// L_2nd ROT R SVD ERR
AND NOT   M0157A	// L_2nd_07 R
AND NOT   M00673	// -
AND NOT   M0157F	// L_2nd_07 R MOVE HOLD
OUT       M01570	// L_2nd_07 R READY
; L108
LOAD      M01570	// L_2nd_07 R READY
TON       T0507 0	// L_2nd_07 R READY
TON       T0707 20	// L_2nd_07 R READY 2s
; L110
LOAD NOT  M0157F	// L_2nd_07 R MOVE HOLD
AND NOT   M0307C	// L_2nd_07 R Pos HOME >
AND NOT   M01571	// L_2nd_07 R POWER ON
NOT
TON       T0607 3000	// L_2nd_07 R NOT MOVE
// output comment: Motor Not Move ¡ÆEAa

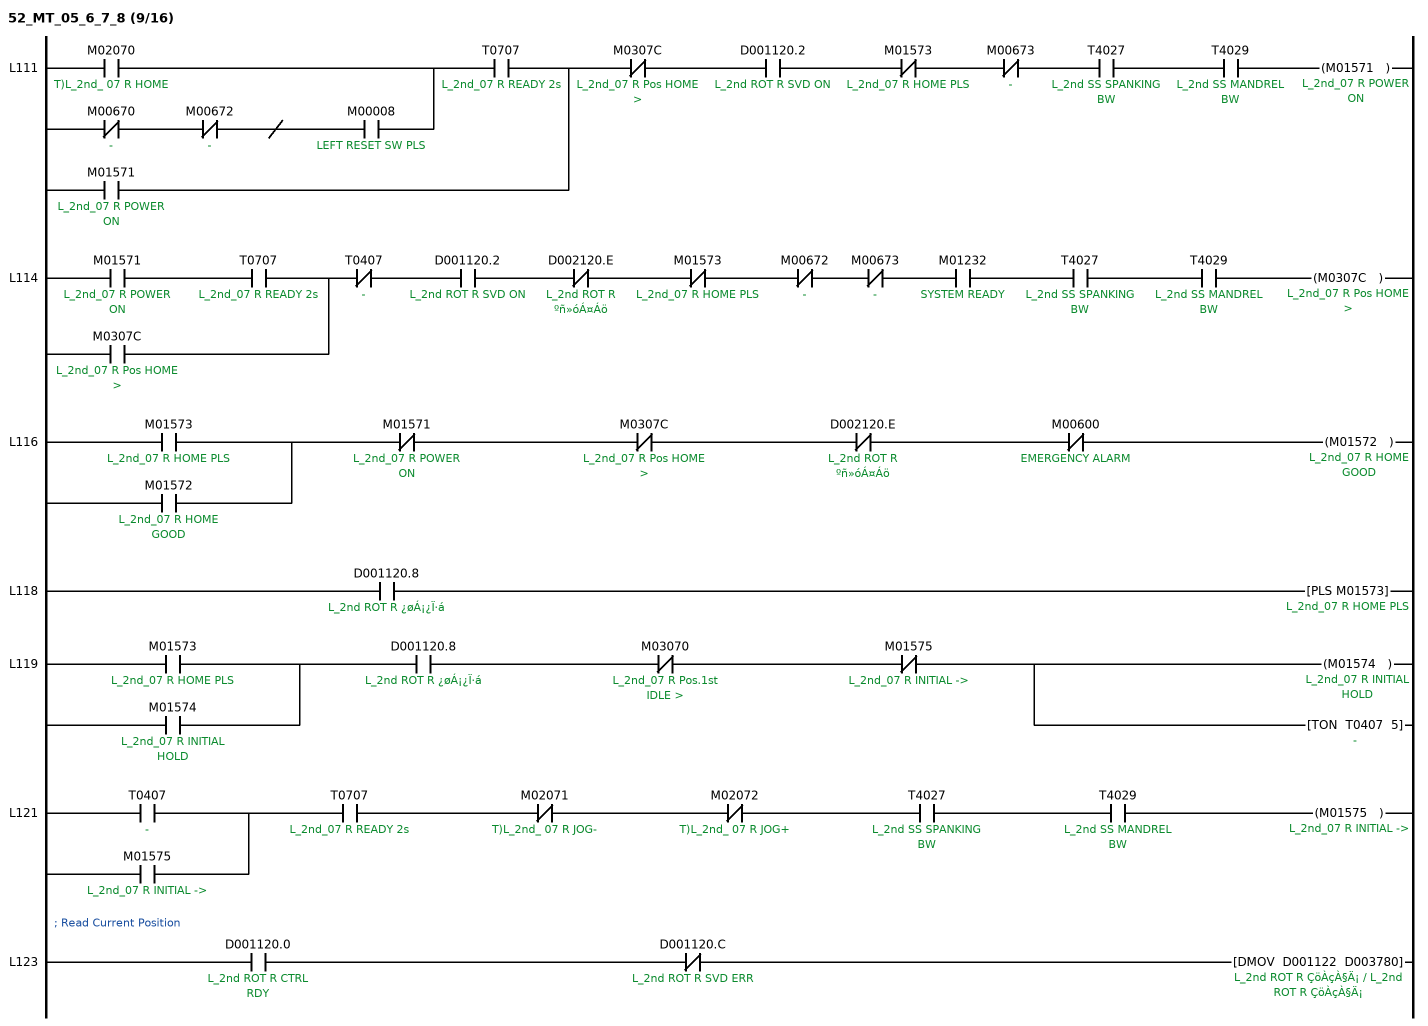
; L111
LOAD      M02070	// T)L_2nd_ 07 R HOME
LOAD NOT  M00670	// -
AND NOT   M00672	// -
NOT
AND       M00008	// LEFT RESET SW PLS
OR LOAD
AND       T0707	// L_2nd_07 R READY 2s
OR        M01571	// L_2nd_07 R POWER ON
AND NOT   M0307C	// L_2nd_07 R Pos HOME >
AND       D001120.2	// L_2nd ROT R SVD ON
AND NOT   M01573	// L_2nd_07 R HOME PLS
AND NOT   M00673	// -
AND       T4027	// L_2nd SS SPANKING BW
AND       T4029	// L_2nd SS MANDREL BW
OUT       M01571	// L_2nd_07 R POWER ON
; L114
LOAD      M01571	// L_2nd_07 R POWER ON
AND       T0707	// L_2nd_07 R READY 2s
OR        M0307C	// L_2nd_07 R Pos HOME >
AND NOT   T0407	// -
AND       D001120.2	// L_2nd ROT R SVD ON
AND NOT   D002120.E	// L_2nd ROT R ºñ»óÁ¤Áö
AND NOT   M01573	// L_2nd_07 R HOME PLS
AND NOT   M00672	// -
AND NOT   M00673	// -
AND       M01232	// SYSTEM READY
AND       T4027	// L_2nd SS SPANKING BW
AND       T4029	// L_2nd SS MANDREL BW
OUT       M0307C	// L_2nd_07 R Pos HOME >
; L116
LOAD      M01573	// L_2nd_07 R HOME PLS
OR        M01572	// L_2nd_07 R HOME GOOD
AND NOT   M01571	// L_2nd_07 R POWER ON
AND NOT   M0307C	// L_2nd_07 R Pos HOME >
AND NOT   D002120.E	// L_2nd ROT R ºñ»óÁ¤Áö
AND NOT   M00600	// EMERGENCY ALARM
OUT       M01572	// L_2nd_07 R HOME GOOD
; L118
LOAD      D001120.8	// L_2nd ROT R ¿øÁ¡¿Ï·á
OUTP      M01573	// L_2nd_07 R HOME PLS
; L119
LOAD      M01573	// L_2nd_07 R HOME PLS
OR        M01574	// L_2nd_07 R INITIAL HOLD
AND       D001120.8	// L_2nd ROT R ¿øÁ¡¿Ï·á
AND NOT   M03070	// L_2nd_07 R Pos.1st IDLE >
AND NOT   M01575	// L_2nd_07 R INITIAL ->
OUT       M01574	// L_2nd_07 R INITIAL HOLD
TON       T0407 5	// -
; L121
LOAD      T0407	// -
OR        M01575	// L_2nd_07 R INITIAL ->
AND       T0707	// L_2nd_07 R READY 2s
AND NOT   M02071	// T)L_2nd_ 07 R JOG-
AND NOT   M02072	// T)L_2nd_ 07 R JOG+
AND       T4027	// L_2nd SS SPANKING BW
AND       T4029	// L_2nd SS MANDREL BW
OUT       M01575	// L_2nd_07 R INITIAL ->
; L123
LOAD      D001120.0	// L_2nd ROT R CTRL RDY
AND NOT   D001120.C	// L_2nd ROT R SVD ERR
DMOV      D001122 D003780	// L_2nd ROT R ÇöÀçÀ§Ä¡ / L_2nd ROT R ÇöÀçÀ§Ä¡
// output comment: Read Current Position

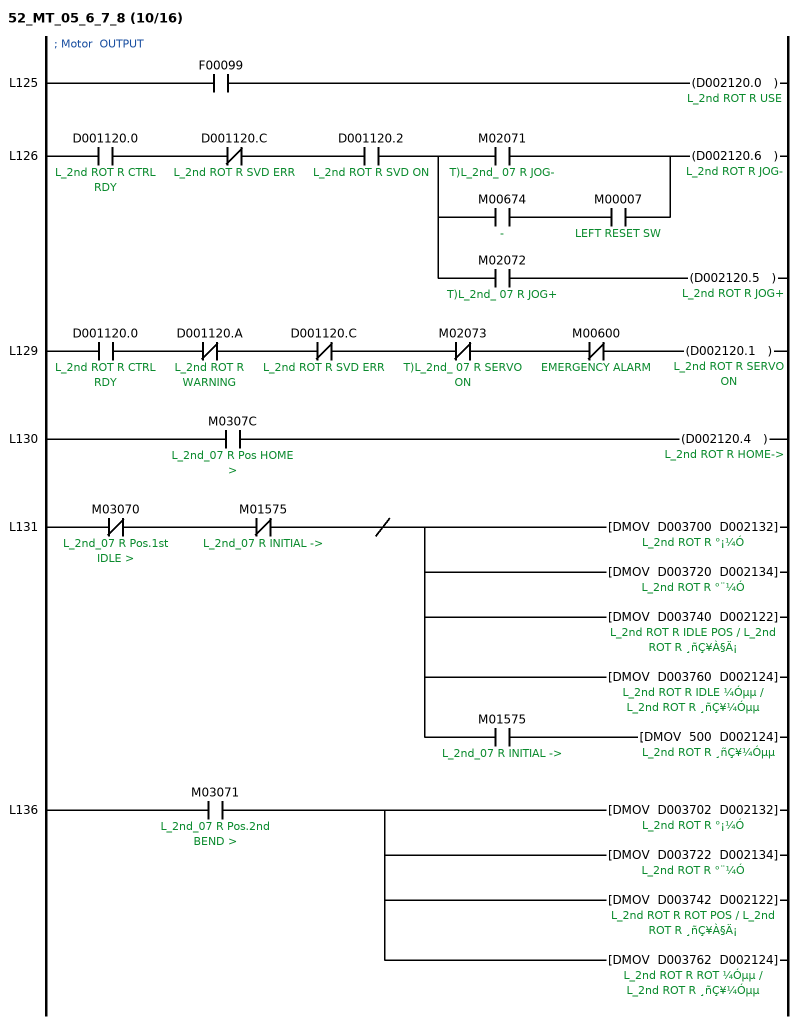
//  Motor  OUTPUT
; L125
LOAD      F00099
OUT       D002120.0	// L_2nd ROT R USE
; L126
LOAD      D001120.0	// L_2nd ROT R CTRL RDY
AND NOT   D001120.C	// L_2nd ROT R SVD ERR
AND       D001120.2	// L_2nd ROT R SVD ON
MPUSH
LOAD      M02071	// T)L_2nd_ 07 R JOG-
LOAD      M00674	// -
AND       M00007	// LEFT RESET SW
OR LOAD
AND LOAD
OUT       D002120.6	// L_2nd ROT R JOG-
MPOP
AND       M02072	// T)L_2nd_ 07 R JOG+
OUT       D002120.5	// L_2nd ROT R JOG+
; L129
LOAD      D001120.0	// L_2nd ROT R CTRL RDY
AND NOT   D001120.A	// L_2nd ROT R WARNING
AND NOT   D001120.C	// L_2nd ROT R SVD ERR
AND NOT   M02073	// T)L_2nd_ 07 R SERVO ON
AND NOT   M00600	// EMERGENCY ALARM
OUT       D002120.1	// L_2nd ROT R SERVO ON
; L130
LOAD      M0307C	// L_2nd_07 R Pos HOME >
OUT       D002120.4	// L_2nd ROT R HOME->
; L131
LOAD NOT  M03070	// L_2nd_07 R Pos.1st IDLE >
AND NOT   M01575	// L_2nd_07 R INITIAL ->
NOT
DMOV      D003700 D002132	// L_2nd ROT R °¡¼Ó
DMOV      D003720 D002134	// L_2nd ROT R °¨¼Ó
DMOV      D003740 D002122	// L_2nd ROT R IDLE POS / L_2nd ROT R ¸ñÇ¥À§Ä¡
DMOV      D003760 D002124	// L_2nd ROT R IDLE ¼Óµµ / L_2nd ROT R ¸ñÇ¥¼Óµµ
AND       M01575	// L_2nd_07 R INITIAL ->
DMOV      500 D002124	// L_2nd ROT R ¸ñÇ¥¼Óµµ
; L136
LOAD      M03071	// L_2nd_07 R Pos.2nd BEND >
DMOV      D003702 D002132	// L_2nd ROT R °¡¼Ó
DMOV      D003722 D002134	// L_2nd ROT R °¨¼Ó
DMOV      D003742 D002122	// L_2nd ROT R ROT POS / L_2nd ROT R ¸ñÇ¥À§Ä¡
DMOV      D003762 D002124	// L_2nd ROT R ROT ¼Óµµ / L_2nd ROT R ¸ñÇ¥¼Óµµ

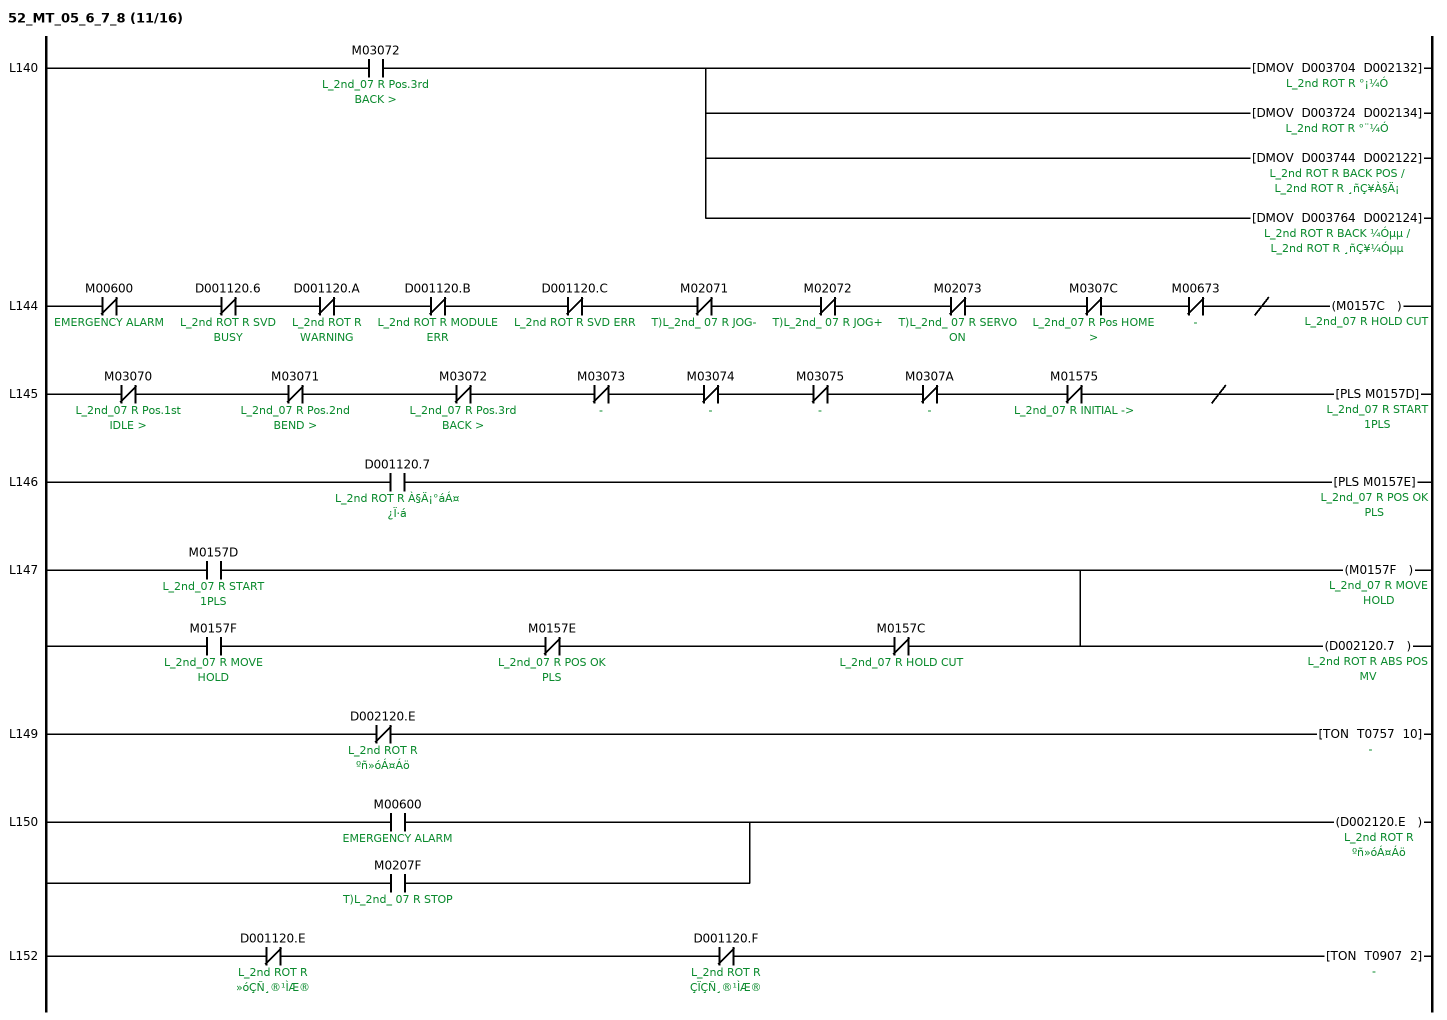
; L140
LOAD      M03072	// L_2nd_07 R Pos.3rd BACK >
DMOV      D003704 D002132	// L_2nd ROT R °¡¼Ó
DMOV      D003724 D002134	// L_2nd ROT R °¨¼Ó
DMOV      D003744 D002122	// L_2nd ROT R BACK POS / L_2nd ROT R ¸ñÇ¥À§Ä¡
DMOV      D003764 D002124	// L_2nd ROT R BACK ¼Óµµ / L_2nd ROT R ¸ñÇ¥¼Óµµ
; L144
LOAD NOT  M00600	// EMERGENCY ALARM
AND NOT   D001120.6	// L_2nd ROT R SVD BUSY
AND NOT   D001120.A	// L_2nd ROT R WARNING
AND NOT   D001120.B	// L_2nd ROT R MODULE ERR
AND NOT   D001120.C	// L_2nd ROT R SVD ERR
AND NOT   M02071	// T)L_2nd_ 07 R JOG-
AND NOT   M02072	// T)L_2nd_ 07 R JOG+
AND NOT   M02073	// T)L_2nd_ 07 R SERVO ON
AND NOT   M0307C	// L_2nd_07 R Pos HOME >
AND NOT   M00673	// -
NOT
OUT       M0157C	// L_2nd_07 R HOLD CUT
; L145
LOAD NOT  M03070	// L_2nd_07 R Pos.1st IDLE >
AND NOT   M03071	// L_2nd_07 R Pos.2nd BEND >
AND NOT   M03072	// L_2nd_07 R Pos.3rd BACK >
AND NOT   M03073	// -
AND NOT   M03074	// -
AND NOT   M03075	// -
AND NOT   M0307A	// -
AND NOT   M01575	// L_2nd_07 R INITIAL ->
NOT
OUTP      M0157D	// L_2nd_07 R START 1PLS
; L146
LOAD      D001120.7	// L_2nd ROT R À§Ä¡°áÁ¤ ¿Ï·á
OUTP      M0157E	// L_2nd_07 R POS OK PLS
; L147
LOAD      M0157D	// L_2nd_07 R START 1PLS
LOAD      M0157F	// L_2nd_07 R MOVE HOLD
AND NOT   M0157E	// L_2nd_07 R POS OK PLS
AND NOT   M0157C	// L_2nd_07 R HOLD CUT
OR LOAD
OUT       M0157F	// L_2nd_07 R MOVE HOLD
OUT       D002120.7	// L_2nd ROT R ABS POS MV
; L149
LOAD NOT  D002120.E	// L_2nd ROT R ºñ»óÁ¤Áö
TON       T0757 10	// -
; L150
LOAD      M00600	// EMERGENCY ALARM
OR        M0207F	// T)L_2nd_ 07 R STOP
OUT       D002120.E	// L_2nd ROT R ºñ»óÁ¤Áö
; L152
LOAD NOT  D001120.E	// L_2nd ROT R »óÇÑ¸®¹ÌÆ®
AND NOT   D001120.F	// L_2nd ROT R ÇÏÇÑ¸®¹ÌÆ®
TON       T0907 2	// -

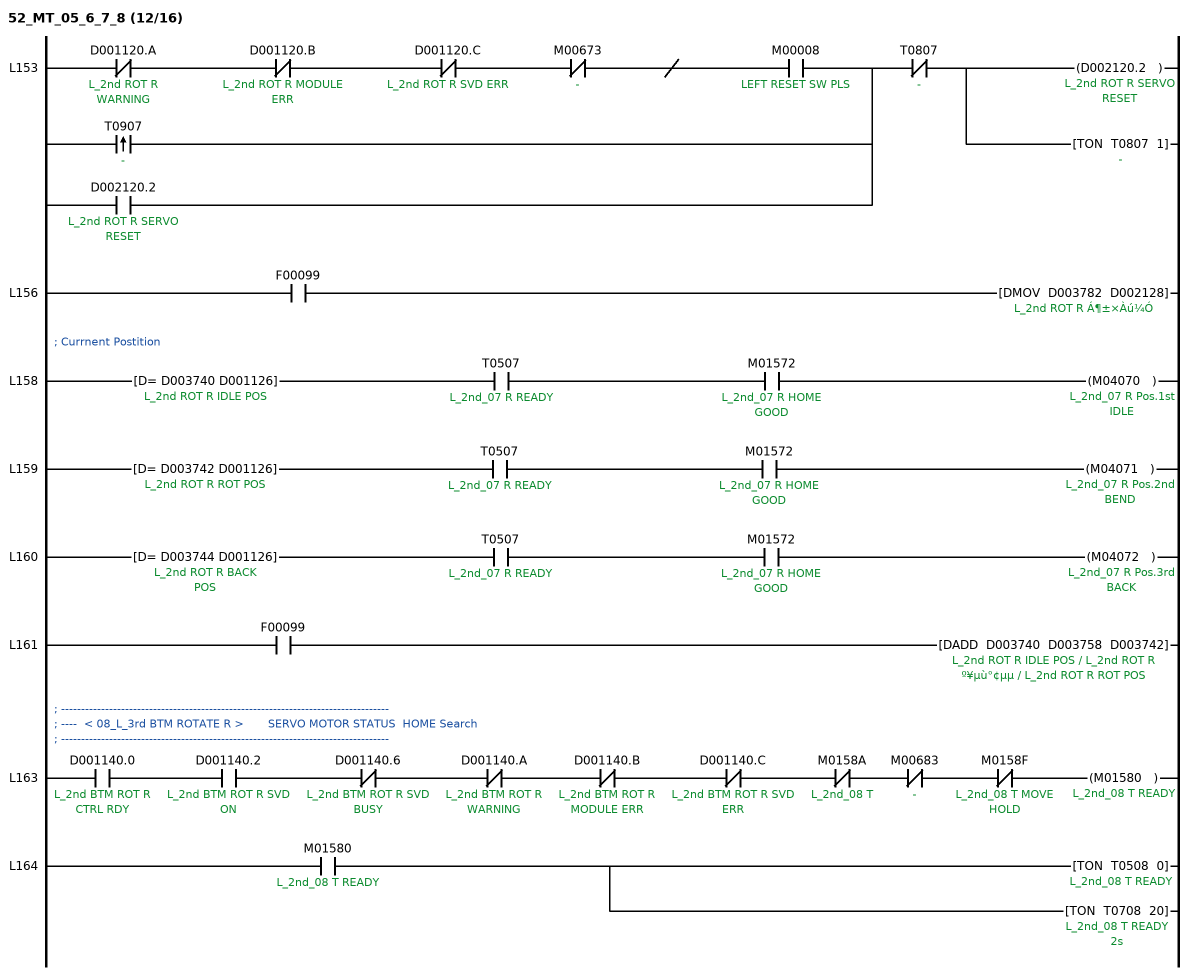
; L153
LOAD NOT  D001120.A	// L_2nd ROT R WARNING
AND NOT   D001120.B	// L_2nd ROT R MODULE ERR
AND NOT   D001120.C	// L_2nd ROT R SVD ERR
AND NOT   M00673	// -
NOT
AND       M00008	// LEFT RESET SW PLS
ORP       T0907	// -
OR        D002120.2	// L_2nd ROT R SERVO RESET
AND NOT   T0807	// -
OUT       D002120.2	// L_2nd ROT R SERVO RESET
TON       T0807 1	// -
; L156
LOAD      F00099
DMOV      D003782 D002128	// L_2nd ROT R Á¶±×Àú¼Ó
// Currnent Postition
; L158
LOADD=    D003740 D001126	// L_2nd ROT R IDLE POS
AND       T0507	// L_2nd_07 R READY
AND       M01572	// L_2nd_07 R HOME GOOD
OUT       M04070	// L_2nd_07 R Pos.1st IDLE
; L159
LOADD=    D003742 D001126	// L_2nd ROT R ROT POS
AND       T0507	// L_2nd_07 R READY
AND       M01572	// L_2nd_07 R HOME GOOD
OUT       M04071	// L_2nd_07 R Pos.2nd BEND
; L160
LOADD=    D003744 D001126	// L_2nd ROT R BACK POS
AND       T0507	// L_2nd_07 R READY
AND       M01572	// L_2nd_07 R HOME GOOD
OUT       M04072	// L_2nd_07 R Pos.3rd BACK
; L161
LOAD      F00099
DADD      D003740 D003758 D003742	// L_2nd ROT R IDLE POS / L_2nd ROT R º¥µù°¢µµ / L_2nd ROT R ROT POS
// ----------------------------------------------------------------------------------
// 
// ----  < 08_L_3rd BTM ROTATE R >       SERVO MOTOR STATUS  HOME Search
// 
// ----------------------------------------------------------------------------------
; L163
LOAD      D001140.0	// L_2nd BTM ROT R CTRL RDY
AND       D001140.2	// L_2nd BTM ROT R SVD ON
AND NOT   D001140.6	// L_2nd BTM ROT R SVD BUSY
AND NOT   D001140.A	// L_2nd BTM ROT R WARNING
AND NOT   D001140.B	// L_2nd BTM ROT R MODULE ERR
AND NOT   D001140.C	// L_2nd BTM ROT R SVD ERR
AND NOT   M0158A	// L_2nd_08 T
AND NOT   M00683	// -
AND NOT   M0158F	// L_2nd_08 T MOVE HOLD
OUT       M01580	// L_2nd_08 T READY
; L164
LOAD      M01580	// L_2nd_08 T READY
TON       T0508 0	// L_2nd_08 T READY
TON       T0708 20	// L_2nd_08 T READY 2s

